(* CODESYS project FengHuang_PackBagbefore_V002.07.18.project

Project tree, tasks and I/O mapping:
  Device : AM403-CPU1608TN, Shenzhen Inovance Control Technology, version 3.5.11.10
      settings: PersistentStartAdddr = 0; PersistentStartEndAddr = 491519; Mode = 1
    application Application
      libraries: Standard, * (System); CmpHCAxisControl, 1.0.2.0 (Inovance); MEGA_Base, 0.0.0.1 (MEGA)
      task MainTask (cyclic, interval 16 ms, priority 1) calls Main
      task EIPSlaveServiceTask (cyclic, interval t#100ms, priority 30) calls EtherNetIPSlave.ServiceCycle
      task ETHERCAT (cyclic, interval 8 ms, priority 0) calls ETHERCAT.EtherCAT_Task, Call_Axis
      task EIPSlaveIOTask (cyclic, interval t#50ms, priority 1) calls EtherNetIPSlave.IOCycle
      DUTS/
        CT/
          data type ST_CT
        IO/
          data type EC6_0032A
          data type EC6_1616_Output
          data type EC6_3200A
          data type EC6_1616_Input
        HMI/
          data type ST_HMI_Vac_Pers
          data type ST_HMI_Cyl_Pers
          data type ST_HMI_Mac_Pers
          data type ST_HMI_Other
          data type ST_HMI_PrgVer
        Machine/
          data type ST_CardtSta
          data type ST_Machine
          data type ST_BagSta
        Data/
          data type ST_Data
        AXIS/
          data type ST_Ethercat
          data type Axis_POS
      FB/
        17_HMIFB/
          function block FB_Proface [ST]: ACT_Control, ACT_Empty, ACT_DummyCheck, ACT_Init
        16_VacuumFB/
          function block FB_Vacuum [ST]: ACT_Manual, ACT_Delay, ACT_Alarm, ACT_Output
        12_BlinkFB/
          data type ST_SysPulse
          function block FB_Blinker [ST]
        14_MachineFB/
          function block FB_Machine_1 [ST]: ACT_status, ACT_CT
          data type ST_OpeButton
          data type ST_DataMachine
          function block FB_Machine [ST]: ACT_Data, ACT_Start, ACT_Pause, ACT_Empty, ACT_Lamp, ACT_CycleTime, ACT_Stop, ACT_Init, ACT_General, ACT_Reset
        10_CylinderFB/
          function block FB_Cylinder [ST]: ACT_Delay, ACT_Output, ACT_Tip, ACT_Manual, ACT_Alarm
        05_StationFB/
          function block FB_Station [ST]: ACT_Init, ACT_State, ACT_Run, ACT_CycleTime, ACT_General
          data type E_State
        50_CycleTime/
          function block FB_CycleTime_2 [ST]
          function block FB_CycleTime_1 [ST]
          function block FB_CycleTime [ST]
        11_AxisFB/
          DUTs/
            data type ST_DataAxis
            data type ST_Axis_REF
          function block FB_Axis [ST]: ACT_Tip, ACT_Move, ACT_Reset, ACT_Halt, ACT_ReinitDrive, ACT_Home, ACT_Stop, ACT_Jog, ACT_Timeout, ACT_Power, ACT_Relative, ACT_InPos, ACT_Velocity, ACT_ReadStatus
      POUS/
        02_STATION/
          program S02_bowlFeeder [ST]: TipAuto, ILC, FlowAuto, TipManual, FlowInit, Alarm, Delay, General
          program S06_OpenBag [ST]: Delay, ILC, Alarm, FlowInit, TipManual, TipAuto, FlowAuto, General
          program S03_takebag [ST]: Delay, TipManual, FlowAuto, ILC, Alarm, General, FlowInit, TipAuto
          program S04_PushCard [ST]: Alarm, FlowInit, TipManual, General, ILC, FlowAuto, TipAuto, Delay
          program Add_distributor [ST]: ILC, Alarm, Delay, TipManual, TipAuto, General, FlowAuto, FlowInit
          program S01_transplant [ST]: TipManual, General, Delay, Alarm, TipAuto, FlowInit, ILC, FlowAuto
          program S05_CircleLine [ST]: Alarm, ILC, TipAuto, TipManual, General, Delay, FlowInit, FlowAuto
        01_LINK/
          program OUTPUT [ST]
          program INPUT [ST]
          program WLTLink [ST]
        03_CALL_standard/
          program ControlMachine [ST]: ACT_ALarm, ACT_Tip, ACT_Try_run, ACT_Count, ACT_InitDone, ACT_EIP_UP
          program Call_Axis [ST]: ACT_Link, ACT_Check
          program CallStandard [ST]: ACT_Machine, ACT_CT, ACT_Proface, ACT_Station, ACT_Blink, ACT_Cylinder, ACT_Vacuum
        program Main [ST]
      GVLS/
        global variables GVL_Standard
        global variables GVL_IO
        global variables GVL_Inside
      Symbols
      FC_check/
        function CheckDivLReal [ST]
        function CheckDivDInt [ST]
        function CheckLRangeUnsigned [ST]
        function CheckDivLInt [ST]
        function CheckRangeUnsigned [ST]
        function CheckRangeSigned [ST]
        function CheckLRangeSigned [ST]
        function CheckBounds [ST]
        function CheckDivReal [ST]
        function CheckPointer [ST]
      global variables PersistentVars
      trace CT (task ETHERCAT, trigger Positive on S05_CircleLine.Axis_Cycleline.rActVelo): S05_CircleLine.Axis_Cycleline.rActVelo
    HardWare Configuration
    ConfigStorage
    Network Configuration
      LocalBus Config
      EtherCAT Config
    Device Diagnosis
    GL10_3200END_1 : AM600-3200END, Inovance, version 00.00.00.10
        settings: ModuleBaseInfoStruct.BusType = 10; ModuleBaseInfoStruct.RackNumber = 1; ModuleBaseInfoStruct.SlotNumber = 2
        unmapped channels: IB(I), IB(II), IB(III), IB(IV)
    HwConfiguratioinDevice : SystemConfig, Inovance, version 00.00.00.10
        settings: NetworkConfigArray.NetworkConfigArray.BusType = 10; NetworkConfigArray.NetworkConfigArray.RackSum = 1; NetworkConfigArray.NetworkConfigArray.HardwareConfigArray.HardwareConfigArray.RackNo = 1; NetworkConfigArray.NetworkConfigArray.HardwareConfigArray.HardwareConfigArray.ModuleNum = 7; NetworkConfigArray.NetworkConfigArray.HardwareConfigArray.HardwareConfigArray.ModuleType.ModuleType = 40899; NetworkConfigArray.NetworkConfigArray.HardwareConfigArray.HardwareConfigArray.ModuleType.ModuleType = 40899; NetworkConfigArray.NetworkConfigArray.HardwareConfigArray.HardwareConfigArray.ModuleType.ModuleType = 40899; NetworkConfigArray.NetworkConfigArray.HardwareConfigArray.HardwareConfigArray.ModuleType.ModuleType = 40899; NetworkConfigArray.NetworkConfigArray.HardwareConfigArray.HardwareConfigArray.ModuleType.ModuleType = 45016; NetworkConfigArray.NetworkConfigArray.HardwareConfigArray.HardwareConfigArray.ModuleType.ModuleType = 45016; NetworkConfigArray.NetworkConfigArray.HardwareConfigArray.HardwareConfigArray.ModuleType.ModuleType = 45016; EnableFun = 1
    MODBUS_TCP : ModbusTCP Device, Inovance, version 00.00.00.10
    HIGH_SPEED_IO : High Speed IO Module, Inovance, version 00.00.00.20
        unmapped channels: InputData, OutputData
      HSIO
    GL10_3200END : AM600-3200END, Inovance, version 00.00.00.10
        settings: ModuleBaseInfoStruct.BusType = 10; ModuleBaseInfoStruct.RackNumber = 1; ModuleBaseInfoStruct.SlotNumber = 1
        unmapped channels: %IB2 IB(I), IB(II), IB(III), IB(IV)
    SoftMotion General Axis Pool
    GL10_0032ETN_1 : AM600-0032ETN, Inovance, version 00.00.00.10
        settings: ModuleBaseInfoStruct.BusType = 10; ModuleBaseInfoStruct.RackNumber = 1; ModuleBaseInfoStruct.SlotNumber = 6
        unmapped channels: QB(I), QB(II), QB(III), QB(IV)
    GL10_0032ETN_2 : AM600-0032ETN, Inovance, version 00.00.00.10
        settings: ModuleBaseInfoStruct.BusType = 10; ModuleBaseInfoStruct.RackNumber = 1; ModuleBaseInfoStruct.SlotNumber = 7
        unmapped channels: QB(I), QB(II), QB(III), QB(IV)
    GL10_3200END_2 : AM600-3200END, Inovance, version 00.00.00.10
        settings: ModuleBaseInfoStruct.BusType = 10; ModuleBaseInfoStruct.RackNumber = 1; ModuleBaseInfoStruct.SlotNumber = 3
        unmapped channels: IB(I), IB(II), IB(III), IB(IV)
    GL10_3200END_3 : AM600-3200END, Inovance, version 00.00.00.10
        settings: ModuleBaseInfoStruct.BusType = 10; ModuleBaseInfoStruct.RackNumber = 1; ModuleBaseInfoStruct.SlotNumber = 4
        unmapped channels: IB(I), IB(II), IB(III), IB(IV)
    GL10_0032ETN : AM600-0032ETN, Inovance, version 00.00.00.10
        settings: ModuleBaseInfoStruct.BusType = 10; ModuleBaseInfoStruct.RackNumber = 1; ModuleBaseInfoStruct.SlotNumber = 5
        unmapped channels: QB(I), QB(II), QB(III), QB(IV)
    ETHERCAT : EtherCAT Master SoftMotion, 3S - Smart Software Solutions GmbH, version 3.5.11.10
        settings:  = 0; MasterCycleTime = 8000; NetworkName = 'eth1'; SelectNetworkByName = TRUE; DisableTaskGeneration = True
      S03_supplybag_Y : SV660_1Axis_00911, Inovance, order no. InoSV660N, version Revision=16#00010000
          settings: FunCodeList = H02;H02-01;H02-02;H03;H03-03;H03-05;; WriteValueList = H02-01_8194_2_1_UINT_RW;H02-02_8194_3_1_UINT_RW;H03-03_8195_4_1_UINT_RW;H03-05_8195_6_1_UINT_RW;; Number of Outputs = 6; Number of Inputs = 10; Number of Infos about Outputs = 6; Number of Infos about Inputs = 10; StationAlias = 1001; Optional = False; DeviceIdenticationADO = 0; DeviceIdenticationMode = 0; Sync.Length = 18; Sync.Length = 32; FMMU.Length = 18; FMMU.Length = 32; AutoUpdate = False; DC sync0 cycletime = 8000; DC sync0 shift time = 0; DC sync1 cycletime = 8000; Number of SDO = 9; Homing method.Index = 16#6098; Homing method.Subindex = 16#00; Homing method.Value = 28; Homing method.Size = 8; Homing method.AbortIfError = FALSE; Homing method.JumpToLine = FALSE; Homing method.Line = 0; Homing method.CompleteAccess = FALSE; Speed during search for switch.Index = 16#6099; Speed during search for switch.Subindex = 16#01; Speed during search for switch.Value = 8388608; Speed during search for switch.Size = 32; Speed during search for switch.AbortIfError = FALSE; Speed during search for switch.JumpToLine = FALSE; Speed during search for switch.Line = 0; Speed during search for switch.CompleteAccess = FALSE; Homing acceleration.Index = 16#609A; Homing acceleration.Subindex = 16#00; Homing acceleration.Value = 419430400; Homing acceleration.Size = 32; Homing acceleration.AbortIfError = FALSE;
            Homing acceleration.JumpToLine = FALSE; Homing acceleration.Line = 0; Homing acceleration.CompleteAccess = FALSE; Speed during search for zero.Index = 16#6099; Speed during search for zero.Subindex = 16#02; Speed during search for zero.Value = 1677722; Speed during search for zero.Size = 32; Speed during search for zero.AbortIfError = FALSE; Speed during search for zero.JumpToLine = FALSE; Speed during search for zero.Line = 0; Speed during search for zero.CompleteAccess = FALSE; Time of home searching.Index = 16#2005; Time of home searching.Subindex = 16#24; Time of home searching.Value = 1500; Time of home searching.Size = 16; Time of home searching.AbortIfError = FALSE; Time of home searching.JumpToLine = FALSE; Time of home searching.Line = 0; Time of home searching.CompleteAccess = FALSE; Positive torque limit value.Index = 16#60E0; Positive torque limit value.Subindex = 16#00; Positive torque limit value.Value = 800; Positive torque limit value.Size = 16; Positive torque limit value.AbortIfError = FALSE; Positive torque limit value.JumpToLine = FALSE; Positive torque limit value.Line = 0; Positive torque limit value.CompleteAccess = FALSE; Negative torque limit value.Index = 16#60E1; Negative torque limit value.Subindex = 16#00; Negative torque limit value.Value = 800; Negative torque limit value.Size = 16; Negative torque limit value.AbortIfError = FALSE; Negative torque limit value.JumpToLine = FALSE; Negative torque limit value.Line = 0; Negative torque limit value.CompleteAccess = FALSE; Max profile velocity.Index = 16#607F; Max profile velocity.Subindex = 16#00; Max profile velocity.Value = 209715200; Max profile velocity.Size = 32; Max profile velocity.AbortIfError = FALSE;
            Max profile velocity.JumpToLine = FALSE; Max profile velocity.Line = 0; Max profile velocity.CompleteAccess = FALSE; RxTxPdo.NumberofEntries = 6; RxTxPdo.Sm = 2; Controlword.Index = 16#6040; Controlword.SubIndex = 0; Controlword.Size = 16; Controlword.DependOnSlot = false; Controlword.DependOnSlotGroup = false; Target position.Index = 16#607A; Target position.SubIndex = 0; Target position.Size = 32; Target position.DependOnSlot = false; Target position.DependOnSlotGroup = false; Touch probe function.Index = 16#60B8; Touch probe function.SubIndex = 0; Touch probe function.Size = 16; Touch probe function.DependOnSlot = false; Touch probe function.DependOnSlotGroup = false; Physical outputs.Index = 16#60FE; Physical outputs.SubIndex = 1; Physical outputs.Size = 32; Physical outputs.DependOnSlot = false; Physical outputs.DependOnSlotGroup = false; Target velocity.Index = 16#60FF; Target velocity.SubIndex = 0; Target velocity.Size = 32; Target velocity.DependOnSlot = false; Target velocity.DependOnSlotGroup = false; Target torque.Index = 16#6071; Target torque.SubIndex = 0; Target torque.Size = 16; Target torque.DependOnSlot = false; Target torque.DependOnSlotGroup = false; RxTxPdo.Sm = -1; RxTxPdo.NumberofEntries = 10; RxTxPdo.Sm = 3; Error code.Index = 16#603F; Error code.SubIndex = 0;
            Error code.Size = 16; Error code.DependOnSlot = false; Error code.DependOnSlotGroup = false; Statusword.Index = 16#6041; Statusword.SubIndex = 0; Statusword.Size = 16; Statusword.DependOnSlot = false; Statusword.DependOnSlotGroup = false; Position actual value.Index = 16#6064; Position actual value.SubIndex = 0; Position actual value.Size = 32; Position actual value.DependOnSlot = false; Position actual value.DependOnSlotGroup = false; Torque actual value.Index = 16#6077; Torque actual value.SubIndex = 0; Torque actual value.Size = 16; Torque actual value.DependOnSlot = false; Torque actual value.DependOnSlotGroup = false; Following error actual value.Index = 16#60F4; Following error actual value.SubIndex = 0; Following error actual value.Size = 32; Following error actual value.DependOnSlot = false; Following error actual value.DependOnSlotGroup = false; Touch probe status.Index = 16#60B9; Touch probe status.SubIndex = 0; Touch probe status.Size = 16; Touch probe status.DependOnSlot = false; Touch probe status.DependOnSlotGroup = false; Touch probe pos1 pos value.Index = 16#60BA; Touch probe pos1 pos value.SubIndex = 0; Touch probe pos1 pos value.Size = 32; Touch probe pos1 pos value.DependOnSlot = false; Touch probe pos1 pos value.DependOnSlotGroup = false; Touch probe pos2 pos value.Index = 16#60BC; Touch probe pos2 pos value.SubIndex = 0; Touch probe pos2 pos value.Size = 32; Touch probe pos2 pos value.DependOnSlot = false; Touch probe pos2 pos value.DependOnSlotGroup = false; Digital inputs.Index = 16#60FD; Digital inputs.SubIndex = 0;
            Digital inputs.Size = 32; Digital inputs.DependOnSlot = false; Digital inputs.DependOnSlotGroup = false; Velocity actual value.Index = 16#606C; Velocity actual value.SubIndex = 0; Velocity actual value.Size = 32; Velocity actual value.DependOnSlot = false; Velocity actual value.DependOnSlotGroup = false; RxTxPdo.Sm = -1; Controlword.Name = 'Controlword'; Controlword.DataType = 'UINT'; Target position.Name = 'Target position'; Target position.DataType = 'DINT'; Touch probe function.Name = 'Touch probe function'; Touch probe function.DataType = 'UINT'; Physical outputs.Name = 'Physical outputs'; Physical outputs.DataType = 'UDINT'; Target velocity.Name = 'Target velocity'; Target velocity.DataType = 'DINT'; Target torque.Name = 'Target torque'; Target torque.DataType = 'INT'; Error code.Name = 'Error code'; Error code.DataType = 'UINT'; Statusword.Name = 'Statusword'; Statusword.DataType = 'UINT'; Position actual value.Name = 'Position actual value'; Position actual value.DataType = 'DINT'; Torque actual value.Name = 'Torque actual value'; Torque actual value.DataType = 'INT'; Following error actual value.Name = 'Following error actual value'; Following error actual value.DataType = 'DINT'; Touch probe status.Name = 'Touch probe status'; Touch probe status.DataType = 'UINT'; Touch probe pos1 pos value.Name = 'Touch probe pos1 pos value'; Touch probe pos1 pos value.DataType = 'DINT'; Touch probe pos2 pos value.Name = 'Touch probe pos2 pos value'; Touch probe pos2 pos value.DataType = 'DINT'; Digital inputs.Name = 'Digital inputs'; Digital inputs.DataType = 'UDINT'; Velocity actual value.Name = 'Velocity actual value';
            Velocity actual value.DataType = 'DINT'
          unmapped channels: %QW500 Controlword, %QD251 Target position, %QW504 Touch probe function, %QD253 Physical outputs, Target velocity, Target torque, %IW500 Error code, %IW501 Statusword, %ID251 Position actual value, Torque actual value, Following error actual value, Touch probe status, Touch probe pos1 pos value, Touch probe pos2 pos value, Digital inputs, Velocity actual value
        Axis_4 : Axis, 3S - Smart Software Solutions GmbH, order no. 0, version 4.0.0.0
            settings: wDriveID = 3; dwRatioTechUnitsDenom = 2097152; iRatioTechUnitsNum = 5; 4000 = 1; 4001 = 0; 4003 = true; 4004 = 25; 4005 = 0; 4006 = 20; 4007 = 1000; 4008 = 4; 4009 = 1500; 4010 = 800; 4011 = 800; 4012 = 500; ScalingIncs = 16#800000; 6005 = 20; AdrOffset_8010 = 1000; BitOffset_8010 = 0; BitLength_8010 = 16; Address_8010 = '%QW500'; Type_8010 = 'UINT'; AddressPointer_8010 = ADR(%QW500); AdrOffset_8020 = 1004; BitOffset_8020 = 0; BitLength_8020 = 32; Address_8020 = '%QD251'; Type_8020 = 'DINT'; AddressPointer_8020 = ADR(%QD251); AdrOffset_8030 = 1016; BitOffset_8030 = 0; BitLength_8030 = 32; Address_8030 = '%QD254'; Type_8030 = 'DINT'; AddressPointer_8030 = ADR(%QD254); AdrOffset_8040 = 1020; BitOffset_8040 = 0; BitLength_8040 = 16; Address_8040 = '%QW510'; Type_8040 = 'INT';
              AddressPointer_8040 = ADR(%QW510); AdrOffset_8050 = 4294967295; BitOffset_8050 = 0; BitLength_8050 = 0; Address_8050 = ''; Type_8050 = ''; AddressPointer_8050 = 0; AdrOffset_8060 = 1008; BitOffset_8060 = 0; BitLength_8060 = 16; Address_8060 = '%QW504'; Type_8060 = 'UINT'; AddressPointer_8060 = ADR(%QW504); AdrOffset_8070 = 4294967295; BitOffset_8070 = 0; BitLength_8070 = 0; Address_8070 = ''; Type_8070 = ''; AddressPointer_8070 = 0; AdrOffset_8080 = 4294967295; BitOffset_8080 = 0; BitLength_8080 = 0; Address_8080 = ''; Type_8080 = ''; AddressPointer_8080 = 0; AdrOffset_8090 = 1012; BitOffset_8090 = 0; BitLength_8090 = 32; Address_8090 = '%QD253'; Type_8090 = 'UDINT'; AddressPointer_8090 = ADR(%QD253); AdrOffset_8510 = 1002; BitOffset_8510 = 0; BitLength_8510 = 16; Address_8510 = '%IW501'; Type_8510 = 'UINT'; AddressPointer_8510 = ADR(%IW501); AdrOffset_8520 = 1004; BitOffset_8520 = 0; BitLength_8520 = 32;
              Address_8520 = '%ID251'; Type_8520 = 'DINT'; AddressPointer_8520 = ADR(%ID251); AdrOffset_8530 = 1032; BitOffset_8530 = 0; BitLength_8530 = 32; Address_8530 = '%ID258'; Type_8530 = 'DINT'; AddressPointer_8530 = ADR(%ID258); AdrOffset_8540 = 1008; BitOffset_8540 = 0; BitLength_8540 = 16; Address_8540 = '%IW504'; Type_8540 = 'INT'; AddressPointer_8540 = ADR(%IW504); AdrOffset_8550 = 4294967295; BitOffset_8550 = 0; BitLength_8550 = 0; Address_8550 = ''; Type_8550 = ''; AddressPointer_8550 = 0; AdrOffset_8560 = 1028; BitOffset_8560 = 0; BitLength_8560 = 32; Address_8560 = '%ID257'; Type_8560 = 'UDINT'; AddressPointer_8560 = ADR(%ID257); AdrOffset_8570 = 1016; BitOffset_8570 = 0; BitLength_8570 = 16; Address_8570 = '%IW508'; Type_8570 = 'UINT'; AddressPointer_8570 = ADR(%IW508); AdrOffset_8580 = 1020; BitOffset_8580 = 0; BitLength_8580 = 32; Address_8580 = '%ID255'; Type_8580 = 'DINT'; AddressPointer_8580 = ADR(%ID255); AdrOffset_8590 = 4294967295;
              BitOffset_8590 = 0; BitLength_8590 = 0; Address_8590 = ''; Type_8590 = ''; AddressPointer_8590 = 0; AdrOffset_8600 = 1024; BitOffset_8600 = 0; BitLength_8600 = 32; Address_8600 = '%ID256'; Type_8600 = 'DINT'; AddressPointer_8600 = ADR(%ID256); AdrOffset_8600 = 4294967295; BitOffset_8600 = 0; BitLength_8600 = 0; Address_8610 = ''; Type_8610 = ''; AddressPointer_8610 = 0; AdrOffset_8620 = 1012; BitOffset_8620 = 0; BitLength_8620 = 32; Address_8620 = '%ID253'; Type_8620 = 'DINT'; AddressPointer_8620 = ADR(%ID253)
      Add_distributor_Y : SV660_1Axis_00911, Inovance, order no. InoSV660N, version Revision=16#00010000
          settings: FunCodeList = H02;H02-01;H03;H03-03;H03-05;; WriteValueList = H02-01_8194_2_1_UINT_RW;H03-03_8195_4_1_UINT_RW;H03-05_8195_6_1_UINT_RW;; Number of Outputs = 6; Number of Inputs = 10; Number of Infos about Outputs = 6; Number of Infos about Inputs = 10; Sync.Length = 18; Sync.Length = 32; FMMU.Length = 18; FMMU.Length = 32; AutoUpdate = False; DC sync0 cycletime = 8000; DC sync1 cycletime = 8000; Number of SDO = 9; Homing method.Index = 16#6098; Homing method.Subindex = 16#00; Homing method.Value = 28; Homing method.Size = 8; Homing method.AbortIfError = FALSE; Homing method.JumpToLine = FALSE; Homing method.Line = 0; Homing method.CompleteAccess = FALSE; Speed during search for switch.Index = 16#6099; Speed during search for switch.Subindex = 16#01; Speed during search for switch.Value = 8388608; Speed during search for switch.Size = 32; Speed during search for switch.AbortIfError = FALSE; Speed during search for switch.JumpToLine = FALSE; Speed during search for switch.Line = 0; Speed during search for switch.CompleteAccess = FALSE; Homing acceleration.Index = 16#609A; Homing acceleration.Subindex = 16#00; Homing acceleration.Value = 419430400; Homing acceleration.Size = 32; Homing acceleration.AbortIfError = FALSE; Homing acceleration.JumpToLine = FALSE; Homing acceleration.Line = 0; Homing acceleration.CompleteAccess = FALSE; Speed during search for zero.Index = 16#6099; Speed during search for zero.Subindex = 16#02;
            Speed during search for zero.Value = 1677722; Speed during search for zero.Size = 32; Speed during search for zero.AbortIfError = FALSE; Speed during search for zero.JumpToLine = FALSE; Speed during search for zero.Line = 0; Speed during search for zero.CompleteAccess = FALSE; Time of home searching.Index = 16#2005; Time of home searching.Subindex = 16#24; Time of home searching.Value = 1500; Time of home searching.Size = 16; Time of home searching.AbortIfError = FALSE; Time of home searching.JumpToLine = FALSE; Time of home searching.Line = 0; Time of home searching.CompleteAccess = FALSE; Positive torque limit value.Index = 16#60E0; Positive torque limit value.Subindex = 16#00; Positive torque limit value.Value = 800; Positive torque limit value.Size = 16; Positive torque limit value.AbortIfError = FALSE; Positive torque limit value.JumpToLine = FALSE; Positive torque limit value.Line = 0; Positive torque limit value.CompleteAccess = FALSE; Negative torque limit value.Index = 16#60E1; Negative torque limit value.Subindex = 16#00; Negative torque limit value.Value = 800; Negative torque limit value.Size = 16; Negative torque limit value.AbortIfError = FALSE; Negative torque limit value.JumpToLine = FALSE; Negative torque limit value.Line = 0; Negative torque limit value.CompleteAccess = FALSE; Max profile velocity.Index = 16#607F; Max profile velocity.Subindex = 16#00; Max profile velocity.Value = 209715200; Max profile velocity.Size = 32; Max profile velocity.AbortIfError = FALSE; Max profile velocity.JumpToLine = FALSE; Max profile velocity.Line = 0; Max profile velocity.CompleteAccess = FALSE; RxTxPdo.NumberofEntries = 6; RxTxPdo.Sm = 2;
            Controlword.Index = 16#6040; Controlword.SubIndex = 0; Controlword.Size = 16; Controlword.DependOnSlot = false; Controlword.DependOnSlotGroup = false; Target position.Index = 16#607A; Target position.SubIndex = 0; Target position.Size = 32; Target position.DependOnSlot = false; Target position.DependOnSlotGroup = false; Touch probe function.Index = 16#60B8; Touch probe function.SubIndex = 0; Touch probe function.Size = 16; Touch probe function.DependOnSlot = false; Touch probe function.DependOnSlotGroup = false; Physical outputs.Index = 16#60FE; Physical outputs.SubIndex = 1; Physical outputs.Size = 32; Physical outputs.DependOnSlot = false; Physical outputs.DependOnSlotGroup = false; Target velocity.Index = 16#60FF; Target velocity.SubIndex = 0; Target velocity.Size = 32; Target velocity.DependOnSlot = false; Target velocity.DependOnSlotGroup = false; Target torque.Index = 16#6071; Target torque.SubIndex = 0; Target torque.Size = 16; Target torque.DependOnSlot = false; Target torque.DependOnSlotGroup = false; RxTxPdo.Sm = -1; RxTxPdo.NumberofEntries = 10; RxTxPdo.Sm = 3; Error code.Index = 16#603F; Error code.SubIndex = 0; Error code.Size = 16; Error code.DependOnSlot = false; Error code.DependOnSlotGroup = false; Statusword.Index = 16#6041; Statusword.SubIndex = 0;
            Statusword.Size = 16; Statusword.DependOnSlot = false; Statusword.DependOnSlotGroup = false; Position actual value.Index = 16#6064; Position actual value.SubIndex = 0; Position actual value.Size = 32; Position actual value.DependOnSlot = false; Position actual value.DependOnSlotGroup = false; Torque actual value.Index = 16#6077; Torque actual value.SubIndex = 0; Torque actual value.Size = 16; Torque actual value.DependOnSlot = false; Torque actual value.DependOnSlotGroup = false; Following error actual value.Index = 16#60F4; Following error actual value.SubIndex = 0; Following error actual value.Size = 32; Following error actual value.DependOnSlot = false; Following error actual value.DependOnSlotGroup = false; Touch probe status.Index = 16#60B9; Touch probe status.SubIndex = 0; Touch probe status.Size = 16; Touch probe status.DependOnSlot = false; Touch probe status.DependOnSlotGroup = false; Touch probe pos1 pos value.Index = 16#60BA; Touch probe pos1 pos value.SubIndex = 0; Touch probe pos1 pos value.Size = 32; Touch probe pos1 pos value.DependOnSlot = false; Touch probe pos1 pos value.DependOnSlotGroup = false; Touch probe pos2 pos value.Index = 16#60BC; Touch probe pos2 pos value.SubIndex = 0; Touch probe pos2 pos value.Size = 32; Touch probe pos2 pos value.DependOnSlot = false; Touch probe pos2 pos value.DependOnSlotGroup = false; Digital inputs.Index = 16#60FD; Digital inputs.SubIndex = 0; Digital inputs.Size = 32; Digital inputs.DependOnSlot = false; Digital inputs.DependOnSlotGroup = false; Velocity actual value.Index = 16#606C; Velocity actual value.SubIndex = 0;
            Velocity actual value.Size = 32; Velocity actual value.DependOnSlot = false; Velocity actual value.DependOnSlotGroup = false; RxTxPdo.Sm = -1; Controlword.Name = 'Controlword'; Controlword.DataType = 'UINT'; Target position.Name = 'Target position'; Target position.DataType = 'DINT'; Touch probe function.Name = 'Touch probe function'; Touch probe function.DataType = 'UINT'; Physical outputs.Name = 'Physical outputs'; Physical outputs.DataType = 'UDINT'; Target velocity.Name = 'Target velocity'; Target velocity.DataType = 'DINT'; Target torque.Name = 'Target torque'; Target torque.DataType = 'INT'; Error code.Name = 'Error code'; Error code.DataType = 'UINT'; Statusword.Name = 'Statusword'; Statusword.DataType = 'UINT'; Position actual value.Name = 'Position actual value'; Position actual value.DataType = 'DINT'; Torque actual value.Name = 'Torque actual value'; Torque actual value.DataType = 'INT'; Following error actual value.Name = 'Following error actual value'; Following error actual value.DataType = 'DINT'; Touch probe status.Name = 'Touch probe status'; Touch probe status.DataType = 'UINT'; Touch probe pos1 pos value.Name = 'Touch probe pos1 pos value'; Touch probe pos1 pos value.DataType = 'DINT'; Touch probe pos2 pos value.Name = 'Touch probe pos2 pos value'; Touch probe pos2 pos value.DataType = 'DINT'; Digital inputs.Name = 'Digital inputs'; Digital inputs.DataType = 'UDINT'; Velocity actual value.Name = 'Velocity actual value'; Velocity actual value.DataType = 'DINT'
          unmapped channels: %QW560 Controlword, Target position, Touch probe function, Physical outputs, Target velocity, Target torque, %IW560 Error code, Statusword, Position actual value, Torque actual value, Following error actual value, Touch probe status, Touch probe pos1 pos value, Touch probe pos2 pos value, Digital inputs, Velocity actual value
        Axis_1 : Axis, 3S - Smart Software Solutions GmbH, order no. 0, version 4.0.0.0
            settings: wDriveID = 0; dwRatioTechUnitsDenom = 2097152; iRatioTechUnitsNum = 5; 4000 = 1; 4001 = 0; 4003 = true; 4004 = 25; 4005 = 0; 4006 = 20; 4007 = 1000; 4008 = 4; 4009 = 1500; 4010 = 800; 4011 = 800; 4012 = 500; ScalingIncs = 16#800000; 6005 = 20; AdrOffset_8010 = 1120; BitOffset_8010 = 0; BitLength_8010 = 16; Address_8010 = '%QW560'; Type_8010 = 'UINT'; AddressPointer_8010 = ADR(%QW560); AdrOffset_8020 = 1124; BitOffset_8020 = 0; BitLength_8020 = 32; Address_8020 = '%QD281'; Type_8020 = 'DINT'; AddressPointer_8020 = ADR(%QD281); AdrOffset_8030 = 1136; BitOffset_8030 = 0; BitLength_8030 = 32; Address_8030 = '%QD284'; Type_8030 = 'DINT'; AddressPointer_8030 = ADR(%QD284); AdrOffset_8040 = 1140; BitOffset_8040 = 0; BitLength_8040 = 16; Address_8040 = '%QW570'; Type_8040 = 'INT';
              AddressPointer_8040 = ADR(%QW570); AdrOffset_8050 = 4294967295; BitOffset_8050 = 0; BitLength_8050 = 0; Address_8050 = ''; Type_8050 = ''; AddressPointer_8050 = 0; AdrOffset_8060 = 1128; BitOffset_8060 = 0; BitLength_8060 = 16; Address_8060 = '%QW564'; Type_8060 = 'UINT'; AddressPointer_8060 = ADR(%QW564); AdrOffset_8070 = 4294967295; BitOffset_8070 = 0; BitLength_8070 = 0; Address_8070 = ''; Type_8070 = ''; AddressPointer_8070 = 0; AdrOffset_8080 = 4294967295; BitOffset_8080 = 0; BitLength_8080 = 0; Address_8080 = ''; Type_8080 = ''; AddressPointer_8080 = 0; AdrOffset_8090 = 1132; BitOffset_8090 = 0; BitLength_8090 = 32; Address_8090 = '%QD283'; Type_8090 = 'UDINT'; AddressPointer_8090 = ADR(%QD283); AdrOffset_8510 = 1122; BitOffset_8510 = 0; BitLength_8510 = 16; Address_8510 = '%IW561'; Type_8510 = 'UINT'; AddressPointer_8510 = ADR(%IW561); AdrOffset_8520 = 1124; BitOffset_8520 = 0; BitLength_8520 = 32;
              Address_8520 = '%ID281'; Type_8520 = 'DINT'; AddressPointer_8520 = ADR(%ID281); AdrOffset_8530 = 1152; BitOffset_8530 = 0; BitLength_8530 = 32; Address_8530 = '%ID288'; Type_8530 = 'DINT'; AddressPointer_8530 = ADR(%ID288); AdrOffset_8540 = 1128; BitOffset_8540 = 0; BitLength_8540 = 16; Address_8540 = '%IW564'; Type_8540 = 'INT'; AddressPointer_8540 = ADR(%IW564); AdrOffset_8550 = 4294967295; BitOffset_8550 = 0; BitLength_8550 = 0; Address_8550 = ''; Type_8550 = ''; AddressPointer_8550 = 0; AdrOffset_8560 = 1148; BitOffset_8560 = 0; BitLength_8560 = 32; Address_8560 = '%ID287'; Type_8560 = 'UDINT'; AddressPointer_8560 = ADR(%ID287); AdrOffset_8570 = 1136; BitOffset_8570 = 0; BitLength_8570 = 16; Address_8570 = '%IW568'; Type_8570 = 'UINT'; AddressPointer_8570 = ADR(%IW568); AdrOffset_8580 = 1140; BitOffset_8580 = 0; BitLength_8580 = 32; Address_8580 = '%ID285'; Type_8580 = 'DINT'; AddressPointer_8580 = ADR(%ID285); AdrOffset_8590 = 4294967295;
              BitOffset_8590 = 0; BitLength_8590 = 0; Address_8590 = ''; Type_8590 = ''; AddressPointer_8590 = 0; AdrOffset_8600 = 1144; BitOffset_8600 = 0; BitLength_8600 = 32; Address_8600 = '%ID286'; Type_8600 = 'DINT'; AddressPointer_8600 = ADR(%ID286); AdrOffset_8600 = 4294967295; BitOffset_8600 = 0; BitLength_8600 = 0; Address_8610 = ''; Type_8610 = ''; AddressPointer_8610 = 0; AdrOffset_8620 = 1132; BitOffset_8620 = 0; BitLength_8620 = 32; Address_8620 = '%ID283'; Type_8620 = 'DINT'; AddressPointer_8620 = ADR(%ID283)
      S03_CycleLine : SV660_1Axis_00911, Inovance, order no. InoSV660N, version Revision=16#00010000
          settings: FunCodeList = H02;H02-02;H0D;H0D-20;; WriteValueList = H02-02_8194_3_0_UINT_RW;H0D-20_8205_21_1_UINT_RW;; Number of Outputs = 6; Number of Inputs = 10; Number of Infos about Outputs = 6; Number of Infos about Inputs = 10; Sync.Length = 18; Sync.Length = 32; FMMU.Length = 18; FMMU.Length = 32; AutoUpdate = False; DC sync0 cycletime = 8000; DC sync1 cycletime = 8000; Number of SDO = 9; Homing method.Index = 16#6098; Homing method.Subindex = 16#00; Homing method.Value = 20; Homing method.Size = 8; Homing method.AbortIfError = FALSE; Homing method.JumpToLine = FALSE; Homing method.Line = 0; Homing method.CompleteAccess = FALSE; Speed during search for switch.Index = 16#6099; Speed during search for switch.Subindex = 16#01; Speed during search for switch.Value = 4194304; Speed during search for switch.Size = 32; Speed during search for switch.AbortIfError = FALSE; Speed during search for switch.JumpToLine = FALSE; Speed during search for switch.Line = 0; Speed during search for switch.CompleteAccess = FALSE; Homing acceleration.Index = 16#609A; Homing acceleration.Subindex = 16#00; Homing acceleration.Value = 209715200; Homing acceleration.Size = 32; Homing acceleration.AbortIfError = FALSE; Homing acceleration.JumpToLine = FALSE; Homing acceleration.Line = 0; Homing acceleration.CompleteAccess = FALSE; Speed during search for zero.Index = 16#6099; Speed during search for zero.Subindex = 16#02;
            Speed during search for zero.Value = 838861; Speed during search for zero.Size = 32; Speed during search for zero.AbortIfError = FALSE; Speed during search for zero.JumpToLine = FALSE; Speed during search for zero.Line = 0; Speed during search for zero.CompleteAccess = FALSE; Time of home searching.Index = 16#2005; Time of home searching.Subindex = 16#24; Time of home searching.Value = 1500; Time of home searching.Size = 16; Time of home searching.AbortIfError = FALSE; Time of home searching.JumpToLine = FALSE; Time of home searching.Line = 0; Time of home searching.CompleteAccess = FALSE; Positive torque limit value.Index = 16#60E0; Positive torque limit value.Subindex = 16#00; Positive torque limit value.Value = 800; Positive torque limit value.Size = 16; Positive torque limit value.AbortIfError = FALSE; Positive torque limit value.JumpToLine = FALSE; Positive torque limit value.Line = 0; Positive torque limit value.CompleteAccess = FALSE; Negative torque limit value.Index = 16#60E1; Negative torque limit value.Subindex = 16#00; Negative torque limit value.Value = 800; Negative torque limit value.Size = 16; Negative torque limit value.AbortIfError = FALSE; Negative torque limit value.JumpToLine = FALSE; Negative torque limit value.Line = 0; Negative torque limit value.CompleteAccess = FALSE; Max profile velocity.Index = 16#607F; Max profile velocity.Subindex = 16#00; Max profile velocity.Value = 104857600; Max profile velocity.Size = 32; Max profile velocity.AbortIfError = FALSE; Max profile velocity.JumpToLine = FALSE; Max profile velocity.Line = 0; Max profile velocity.CompleteAccess = FALSE; RxTxPdo.NumberofEntries = 6; RxTxPdo.Sm = 2;
            Controlword.Index = 16#6040; Controlword.SubIndex = 0; Controlword.Size = 16; Controlword.DependOnSlot = false; Controlword.DependOnSlotGroup = false; Target position.Index = 16#607A; Target position.SubIndex = 0; Target position.Size = 32; Target position.DependOnSlot = false; Target position.DependOnSlotGroup = false; Touch probe function.Index = 16#60B8; Touch probe function.SubIndex = 0; Touch probe function.Size = 16; Touch probe function.DependOnSlot = false; Touch probe function.DependOnSlotGroup = false; Physical outputs.Index = 16#60FE; Physical outputs.SubIndex = 1; Physical outputs.Size = 32; Physical outputs.DependOnSlot = false; Physical outputs.DependOnSlotGroup = false; Target velocity.Index = 16#60FF; Target velocity.SubIndex = 0; Target velocity.Size = 32; Target velocity.DependOnSlot = false; Target velocity.DependOnSlotGroup = false; Target torque.Index = 16#6071; Target torque.SubIndex = 0; Target torque.Size = 16; Target torque.DependOnSlot = false; Target torque.DependOnSlotGroup = false; RxTxPdo.Sm = -1; RxTxPdo.NumberofEntries = 10; RxTxPdo.Sm = 3; Error code.Index = 16#603F; Error code.SubIndex = 0; Error code.Size = 16; Error code.DependOnSlot = false; Error code.DependOnSlotGroup = false; Statusword.Index = 16#6041; Statusword.SubIndex = 0;
            Statusword.Size = 16; Statusword.DependOnSlot = false; Statusword.DependOnSlotGroup = false; Position actual value.Index = 16#6064; Position actual value.SubIndex = 0; Position actual value.Size = 32; Position actual value.DependOnSlot = false; Position actual value.DependOnSlotGroup = false; Torque actual value.Index = 16#6077; Torque actual value.SubIndex = 0; Torque actual value.Size = 16; Torque actual value.DependOnSlot = false; Torque actual value.DependOnSlotGroup = false; Following error actual value.Index = 16#60F4; Following error actual value.SubIndex = 0; Following error actual value.Size = 32; Following error actual value.DependOnSlot = false; Following error actual value.DependOnSlotGroup = false; Touch probe status.Index = 16#60B9; Touch probe status.SubIndex = 0; Touch probe status.Size = 16; Touch probe status.DependOnSlot = false; Touch probe status.DependOnSlotGroup = false; Touch probe pos1 pos value.Index = 16#60BA; Touch probe pos1 pos value.SubIndex = 0; Touch probe pos1 pos value.Size = 32; Touch probe pos1 pos value.DependOnSlot = false; Touch probe pos1 pos value.DependOnSlotGroup = false; Touch probe pos2 pos value.Index = 16#60BC; Touch probe pos2 pos value.SubIndex = 0; Touch probe pos2 pos value.Size = 32; Touch probe pos2 pos value.DependOnSlot = false; Touch probe pos2 pos value.DependOnSlotGroup = false; Digital inputs.Index = 16#60FD; Digital inputs.SubIndex = 0; Digital inputs.Size = 32; Digital inputs.DependOnSlot = false; Digital inputs.DependOnSlotGroup = false; Velocity actual value.Index = 16#606C; Velocity actual value.SubIndex = 0;
            Velocity actual value.Size = 32; Velocity actual value.DependOnSlot = false; Velocity actual value.DependOnSlotGroup = false; RxTxPdo.Sm = -1; Controlword.Name = 'Controlword'; Controlword.DataType = 'UINT'; Target position.Name = 'Target position'; Target position.DataType = 'DINT'; Touch probe function.Name = 'Touch probe function'; Touch probe function.DataType = 'UINT'; Physical outputs.Name = 'Physical outputs'; Physical outputs.DataType = 'UDINT'; Target velocity.Name = 'Target velocity'; Target velocity.DataType = 'DINT'; Target torque.Name = 'Target torque'; Target torque.DataType = 'INT'; Error code.Name = 'Error code'; Error code.DataType = 'UINT'; Statusword.Name = 'Statusword'; Statusword.DataType = 'UINT'; Position actual value.Name = 'Position actual value'; Position actual value.DataType = 'DINT'; Torque actual value.Name = 'Torque actual value'; Torque actual value.DataType = 'INT'; Following error actual value.Name = 'Following error actual value'; Following error actual value.DataType = 'DINT'; Touch probe status.Name = 'Touch probe status'; Touch probe status.DataType = 'UINT'; Touch probe pos1 pos value.Name = 'Touch probe pos1 pos value'; Touch probe pos1 pos value.DataType = 'DINT'; Touch probe pos2 pos value.Name = 'Touch probe pos2 pos value'; Touch probe pos2 pos value.DataType = 'DINT'; Digital inputs.Name = 'Digital inputs'; Digital inputs.DataType = 'UDINT'; Velocity actual value.Name = 'Velocity actual value'; Velocity actual value.DataType = 'DINT'
          unmapped channels: %QW600 Controlword, Target position, Touch probe function, Physical outputs, Target velocity, Target torque, %IW600 Error code, Statusword, Position actual value, Torque actual value, Following error actual value, Touch probe status, Touch probe pos1 pos value, Touch probe pos2 pos value, Digital inputs, Velocity actual value
        Axis_3 : Axis, 3S - Smart Software Solutions GmbH, order no. 0, version 4.0.0.0
            settings: wDriveID = 2; dwRatioTechUnitsDenom = 1048576; iRatioTechUnitsNum = 5; 4000 = 1; 4001 = 1; 4003 = true; 4004 = 17; 4005 = 0; 4006 = 20; 4007 = 1000; 4008 = 4; 4009 = 1500; 4010 = 800; 4011 = 800; 4012 = 500; ScalingIncs = 16#800000; ScalingMotorTurns2 = 5; 6005 = 200; AdrOffset_8010 = 1200; BitOffset_8010 = 0; BitLength_8010 = 16; Address_8010 = '%QW600'; Type_8010 = 'UINT'; AddressPointer_8010 = ADR(%QW600); AdrOffset_8020 = 1204; BitOffset_8020 = 0; BitLength_8020 = 32; Address_8020 = '%QD301'; Type_8020 = 'DINT'; AddressPointer_8020 = ADR(%QD301); AdrOffset_8030 = 1216; BitOffset_8030 = 0; BitLength_8030 = 32; Address_8030 = '%QD304'; Type_8030 = 'DINT'; AddressPointer_8030 = ADR(%QD304); AdrOffset_8040 = 1220; BitOffset_8040 = 0; BitLength_8040 = 16; Address_8040 = '%QW610';
              Type_8040 = 'INT'; AddressPointer_8040 = ADR(%QW610); AdrOffset_8050 = 4294967295; BitOffset_8050 = 0; BitLength_8050 = 0; Address_8050 = ''; Type_8050 = ''; AddressPointer_8050 = 0; AdrOffset_8060 = 1208; BitOffset_8060 = 0; BitLength_8060 = 16; Address_8060 = '%QW604'; Type_8060 = 'UINT'; AddressPointer_8060 = ADR(%QW604); AdrOffset_8070 = 4294967295; BitOffset_8070 = 0; BitLength_8070 = 0; Address_8070 = ''; Type_8070 = ''; AddressPointer_8070 = 0; AdrOffset_8080 = 4294967295; BitOffset_8080 = 0; BitLength_8080 = 0; Address_8080 = ''; Type_8080 = ''; AddressPointer_8080 = 0; AdrOffset_8090 = 1212; BitOffset_8090 = 0; BitLength_8090 = 32; Address_8090 = '%QD303'; Type_8090 = 'UDINT'; AddressPointer_8090 = ADR(%QD303); AdrOffset_8510 = 1202; BitOffset_8510 = 0; BitLength_8510 = 16; Address_8510 = '%IW601'; Type_8510 = 'UINT'; AddressPointer_8510 = ADR(%IW601); AdrOffset_8520 = 1204; BitOffset_8520 = 0;
              BitLength_8520 = 32; Address_8520 = '%ID301'; Type_8520 = 'DINT'; AddressPointer_8520 = ADR(%ID301); AdrOffset_8530 = 1232; BitOffset_8530 = 0; BitLength_8530 = 32; Address_8530 = '%ID308'; Type_8530 = 'DINT'; AddressPointer_8530 = ADR(%ID308); AdrOffset_8540 = 1208; BitOffset_8540 = 0; BitLength_8540 = 16; Address_8540 = '%IW604'; Type_8540 = 'INT'; AddressPointer_8540 = ADR(%IW604); AdrOffset_8550 = 4294967295; BitOffset_8550 = 0; BitLength_8550 = 0; Address_8550 = ''; Type_8550 = ''; AddressPointer_8550 = 0; AdrOffset_8560 = 1228; BitOffset_8560 = 0; BitLength_8560 = 32; Address_8560 = '%ID307'; Type_8560 = 'UDINT'; AddressPointer_8560 = ADR(%ID307); AdrOffset_8570 = 1216; BitOffset_8570 = 0; BitLength_8570 = 16; Address_8570 = '%IW608'; Type_8570 = 'UINT'; AddressPointer_8570 = ADR(%IW608); AdrOffset_8580 = 1220; BitOffset_8580 = 0; BitLength_8580 = 32; Address_8580 = '%ID305'; Type_8580 = 'DINT'; AddressPointer_8580 = ADR(%ID305);
              AdrOffset_8590 = 4294967295; BitOffset_8590 = 0; BitLength_8590 = 0; Address_8590 = ''; Type_8590 = ''; AddressPointer_8590 = 0; AdrOffset_8600 = 1224; BitOffset_8600 = 0; BitLength_8600 = 32; Address_8600 = '%ID306'; Type_8600 = 'DINT'; AddressPointer_8600 = ADR(%ID306); AdrOffset_8600 = 4294967295; BitOffset_8600 = 0; BitLength_8600 = 0; Address_8610 = ''; Type_8610 = ''; AddressPointer_8610 = 0; AdrOffset_8620 = 1212; BitOffset_8620 = 0; BitLength_8620 = 32; Address_8620 = '%ID303'; Type_8620 = 'DINT'; AddressPointer_8620 = ADR(%ID303)
      S01_CycleLine : SV660_1Axis_00911, Inovance, order no. InoSV660N, version Revision=16#00010000
          settings: FunCodeList = H02;H02-02;H03;H03-03;H03-05;H0D;H0D-20;; WriteValueList = H02-02_8194_3_1_UINT_RW;H03-03_8195_4_0_UINT_RW;H03-05_8195_6_0_UINT_RW;H0D-20_8205_21_0_UINT_RW;; Number of Outputs = 6; Number of Inputs = 10; Number of Infos about Outputs = 6; Number of Infos about Inputs = 10; Sync.Length = 18; Sync.Length = 32; FMMU.Length = 18; FMMU.Length = 32; AutoUpdate = False; DC sync0 cycletime = 8000; DC sync1 cycletime = 8000; Number of SDO = 9; Homing method.Index = 16#6098; Homing method.Subindex = 16#00; Homing method.Value = 20; Homing method.Size = 8; Homing method.AbortIfError = FALSE; Homing method.JumpToLine = FALSE; Homing method.Line = 0; Homing method.CompleteAccess = FALSE; Speed during search for switch.Index = 16#6099; Speed during search for switch.Subindex = 16#01; Speed during search for switch.Value = 4194304; Speed during search for switch.Size = 32; Speed during search for switch.AbortIfError = FALSE; Speed during search for switch.JumpToLine = FALSE; Speed during search for switch.Line = 0; Speed during search for switch.CompleteAccess = FALSE; Homing acceleration.Index = 16#609A; Homing acceleration.Subindex = 16#00; Homing acceleration.Value = 209715200; Homing acceleration.Size = 32; Homing acceleration.AbortIfError = FALSE; Homing acceleration.JumpToLine = FALSE; Homing acceleration.Line = 0; Homing acceleration.CompleteAccess = FALSE; Speed during search for zero.Index = 16#6099; Speed during search for zero.Subindex = 16#02;
            Speed during search for zero.Value = 838861; Speed during search for zero.Size = 32; Speed during search for zero.AbortIfError = FALSE; Speed during search for zero.JumpToLine = FALSE; Speed during search for zero.Line = 0; Speed during search for zero.CompleteAccess = FALSE; Time of home searching.Index = 16#2005; Time of home searching.Subindex = 16#24; Time of home searching.Value = 1500; Time of home searching.Size = 16; Time of home searching.AbortIfError = FALSE; Time of home searching.JumpToLine = FALSE; Time of home searching.Line = 0; Time of home searching.CompleteAccess = FALSE; Positive torque limit value.Index = 16#60E0; Positive torque limit value.Subindex = 16#00; Positive torque limit value.Value = 800; Positive torque limit value.Size = 16; Positive torque limit value.AbortIfError = FALSE; Positive torque limit value.JumpToLine = FALSE; Positive torque limit value.Line = 0; Positive torque limit value.CompleteAccess = FALSE; Negative torque limit value.Index = 16#60E1; Negative torque limit value.Subindex = 16#00; Negative torque limit value.Value = 800; Negative torque limit value.Size = 16; Negative torque limit value.AbortIfError = FALSE; Negative torque limit value.JumpToLine = FALSE; Negative torque limit value.Line = 0; Negative torque limit value.CompleteAccess = FALSE; Max profile velocity.Index = 16#607F; Max profile velocity.Subindex = 16#00; Max profile velocity.Value = 104857600; Max profile velocity.Size = 32; Max profile velocity.AbortIfError = FALSE; Max profile velocity.JumpToLine = FALSE; Max profile velocity.Line = 0; Max profile velocity.CompleteAccess = FALSE; RxTxPdo.NumberofEntries = 6; RxTxPdo.Sm = 2;
            Controlword.Index = 16#6040; Controlword.SubIndex = 0; Controlword.Size = 16; Controlword.DependOnSlot = false; Controlword.DependOnSlotGroup = false; Target position.Index = 16#607A; Target position.SubIndex = 0; Target position.Size = 32; Target position.DependOnSlot = false; Target position.DependOnSlotGroup = false; Touch probe function.Index = 16#60B8; Touch probe function.SubIndex = 0; Touch probe function.Size = 16; Touch probe function.DependOnSlot = false; Touch probe function.DependOnSlotGroup = false; Physical outputs.Index = 16#60FE; Physical outputs.SubIndex = 1; Physical outputs.Size = 32; Physical outputs.DependOnSlot = false; Physical outputs.DependOnSlotGroup = false; Target velocity.Index = 16#60FF; Target velocity.SubIndex = 0; Target velocity.Size = 32; Target velocity.DependOnSlot = false; Target velocity.DependOnSlotGroup = false; Target torque.Index = 16#6071; Target torque.SubIndex = 0; Target torque.Size = 16; Target torque.DependOnSlot = false; Target torque.DependOnSlotGroup = false; RxTxPdo.Sm = -1; RxTxPdo.NumberofEntries = 10; RxTxPdo.Sm = 3; Error code.Index = 16#603F; Error code.SubIndex = 0; Error code.Size = 16; Error code.DependOnSlot = false; Error code.DependOnSlotGroup = false; Statusword.Index = 16#6041; Statusword.SubIndex = 0;
            Statusword.Size = 16; Statusword.DependOnSlot = false; Statusword.DependOnSlotGroup = false; Position actual value.Index = 16#6064; Position actual value.SubIndex = 0; Position actual value.Size = 32; Position actual value.DependOnSlot = false; Position actual value.DependOnSlotGroup = false; Torque actual value.Index = 16#6077; Torque actual value.SubIndex = 0; Torque actual value.Size = 16; Torque actual value.DependOnSlot = false; Torque actual value.DependOnSlotGroup = false; Following error actual value.Index = 16#60F4; Following error actual value.SubIndex = 0; Following error actual value.Size = 32; Following error actual value.DependOnSlot = false; Following error actual value.DependOnSlotGroup = false; Touch probe status.Index = 16#60B9; Touch probe status.SubIndex = 0; Touch probe status.Size = 16; Touch probe status.DependOnSlot = false; Touch probe status.DependOnSlotGroup = false; Touch probe pos1 pos value.Index = 16#60BA; Touch probe pos1 pos value.SubIndex = 0; Touch probe pos1 pos value.Size = 32; Touch probe pos1 pos value.DependOnSlot = false; Touch probe pos1 pos value.DependOnSlotGroup = false; Touch probe pos2 pos value.Index = 16#60BC; Touch probe pos2 pos value.SubIndex = 0; Touch probe pos2 pos value.Size = 32; Touch probe pos2 pos value.DependOnSlot = false; Touch probe pos2 pos value.DependOnSlotGroup = false; Digital inputs.Index = 16#60FD; Digital inputs.SubIndex = 0; Digital inputs.Size = 32; Digital inputs.DependOnSlot = false; Digital inputs.DependOnSlotGroup = false; Velocity actual value.Index = 16#606C; Velocity actual value.SubIndex = 0;
            Velocity actual value.Size = 32; Velocity actual value.DependOnSlot = false; Velocity actual value.DependOnSlotGroup = false; RxTxPdo.Sm = -1; Controlword.Name = 'Controlword'; Controlword.DataType = 'UINT'; Target position.Name = 'Target position'; Target position.DataType = 'DINT'; Touch probe function.Name = 'Touch probe function'; Touch probe function.DataType = 'UINT'; Physical outputs.Name = 'Physical outputs'; Physical outputs.DataType = 'UDINT'; Target velocity.Name = 'Target velocity'; Target velocity.DataType = 'DINT'; Target torque.Name = 'Target torque'; Target torque.DataType = 'INT'; Error code.Name = 'Error code'; Error code.DataType = 'UINT'; Statusword.Name = 'Statusword'; Statusword.DataType = 'UINT'; Position actual value.Name = 'Position actual value'; Position actual value.DataType = 'DINT'; Torque actual value.Name = 'Torque actual value'; Torque actual value.DataType = 'INT'; Following error actual value.Name = 'Following error actual value'; Following error actual value.DataType = 'DINT'; Touch probe status.Name = 'Touch probe status'; Touch probe status.DataType = 'UINT'; Touch probe pos1 pos value.Name = 'Touch probe pos1 pos value'; Touch probe pos1 pos value.DataType = 'DINT'; Touch probe pos2 pos value.Name = 'Touch probe pos2 pos value'; Touch probe pos2 pos value.DataType = 'DINT'; Digital inputs.Name = 'Digital inputs'; Digital inputs.DataType = 'UDINT'; Velocity actual value.Name = 'Velocity actual value'; Velocity actual value.DataType = 'DINT'
          unmapped channels: %QW580 Controlword, Target position, Touch probe function, Physical outputs, Target velocity, Target torque, %IW580 Error code, Statusword, Position actual value, Torque actual value, Following error actual value, Touch probe status, Touch probe pos1 pos value, Touch probe pos2 pos value, Digital inputs, Velocity actual value
        Axis_2 : Axis, 3S - Smart Software Solutions GmbH, order no. 0, version 4.0.0.0
            settings: dwRatioTechUnitsDenom = 1048576; iRatioTechUnitsNum = 5; 4000 = 1; 4001 = 1; 4003 = true; 4004 = 17; 4005 = 0; 4006 = 20; 4007 = 1000; 4008 = 4; 4009 = 1500; 4010 = 800; 4011 = 800; 4012 = 500; ScalingIncs = 16#800000; ScalingMotorTurns2 = 5; 6005 = 200; AdrOffset_8010 = 1160; BitOffset_8010 = 0; BitLength_8010 = 16; Address_8010 = '%QW580'; Type_8010 = 'UINT'; AddressPointer_8010 = ADR(%QW580); AdrOffset_8020 = 1164; BitOffset_8020 = 0; BitLength_8020 = 32; Address_8020 = '%QD291'; Type_8020 = 'DINT'; AddressPointer_8020 = ADR(%QD291); AdrOffset_8030 = 1176; BitOffset_8030 = 0; BitLength_8030 = 32; Address_8030 = '%QD294'; Type_8030 = 'DINT'; AddressPointer_8030 = ADR(%QD294); AdrOffset_8040 = 1180; BitOffset_8040 = 0; BitLength_8040 = 16; Address_8040 = '%QW590'; Type_8040 = 'INT';
              AddressPointer_8040 = ADR(%QW590); AdrOffset_8050 = 4294967295; BitOffset_8050 = 0; BitLength_8050 = 0; Address_8050 = ''; Type_8050 = ''; AddressPointer_8050 = 0; AdrOffset_8060 = 1168; BitOffset_8060 = 0; BitLength_8060 = 16; Address_8060 = '%QW584'; Type_8060 = 'UINT'; AddressPointer_8060 = ADR(%QW584); AdrOffset_8070 = 4294967295; BitOffset_8070 = 0; BitLength_8070 = 0; Address_8070 = ''; Type_8070 = ''; AddressPointer_8070 = 0; AdrOffset_8080 = 4294967295; BitOffset_8080 = 0; BitLength_8080 = 0; Address_8080 = ''; Type_8080 = ''; AddressPointer_8080 = 0; AdrOffset_8090 = 1172; BitOffset_8090 = 0; BitLength_8090 = 32; Address_8090 = '%QD293'; Type_8090 = 'UDINT'; AddressPointer_8090 = ADR(%QD293); AdrOffset_8510 = 1162; BitOffset_8510 = 0; BitLength_8510 = 16; Address_8510 = '%IW581'; Type_8510 = 'UINT'; AddressPointer_8510 = ADR(%IW581); AdrOffset_8520 = 1164; BitOffset_8520 = 0; BitLength_8520 = 32;
              Address_8520 = '%ID291'; Type_8520 = 'DINT'; AddressPointer_8520 = ADR(%ID291); AdrOffset_8530 = 1192; BitOffset_8530 = 0; BitLength_8530 = 32; Address_8530 = '%ID298'; Type_8530 = 'DINT'; AddressPointer_8530 = ADR(%ID298); AdrOffset_8540 = 1168; BitOffset_8540 = 0; BitLength_8540 = 16; Address_8540 = '%IW584'; Type_8540 = 'INT'; AddressPointer_8540 = ADR(%IW584); AdrOffset_8550 = 4294967295; BitOffset_8550 = 0; BitLength_8550 = 0; Address_8550 = ''; Type_8550 = ''; AddressPointer_8550 = 0; AdrOffset_8560 = 1188; BitOffset_8560 = 0; BitLength_8560 = 32; Address_8560 = '%ID297'; Type_8560 = 'UDINT'; AddressPointer_8560 = ADR(%ID297); AdrOffset_8570 = 1176; BitOffset_8570 = 0; BitLength_8570 = 16; Address_8570 = '%IW588'; Type_8570 = 'UINT'; AddressPointer_8570 = ADR(%IW588); AdrOffset_8580 = 1180; BitOffset_8580 = 0; BitLength_8580 = 32; Address_8580 = '%ID295'; Type_8580 = 'DINT'; AddressPointer_8580 = ADR(%ID295); AdrOffset_8590 = 4294967295;
              BitOffset_8590 = 0; BitLength_8590 = 0; Address_8590 = ''; Type_8590 = ''; AddressPointer_8590 = 0; AdrOffset_8600 = 1184; BitOffset_8600 = 0; BitLength_8600 = 32; Address_8600 = '%ID296'; Type_8600 = 'DINT'; AddressPointer_8600 = ADR(%ID296); AdrOffset_8600 = 4294967295; BitOffset_8600 = 0; BitLength_8600 = 0; Address_8610 = ''; Type_8610 = ''; AddressPointer_8610 = 0; AdrOffset_8620 = 1172; BitOffset_8620 = 0; BitLength_8620 = 32; Address_8620 = '%ID293'; Type_8620 = 'DINT'; AddressPointer_8620 = ADR(%ID293)
      S02_PPU_Module : CL3-EC808AC(COE), Leadshine Technology Co.,Ltd., order no. CL3-EC808AC, version Revision=16#00000001
          settings: AutoUpdate = False; DC sync0 cycletime = 8000; DC sync1 cycletime = 8000; Number of SDO = 5; Homing Velocity (fast).Index = 16#6099; Homing Velocity (fast).Subindex = 16#01; Homing Velocity (fast).Value = 2000; Homing Velocity (fast).Size = 32; Homing Velocity (fast).AbortIfError = FALSE; Homing Velocity (fast).JumpToLine = FALSE; Homing Velocity (fast).Line = 0; Homing Velocity (fast).CompleteAccess = False; Homing Acceleration.Index = 16#609A; Homing Acceleration.Subindex = 16#00; Homing Acceleration.Value = 5000; Homing Acceleration.Size = 32; Homing Acceleration.AbortIfError = FALSE; Homing Acceleration.JumpToLine = FALSE; Homing Acceleration.Line = 0; Homing Acceleration.CompleteAccess = False; Homing Velocity (slow).Index = 16#6099; Homing Velocity (slow).Subindex = 16#02; Homing Velocity (slow).Value = 100; Homing Velocity (slow).Size = 32; Homing Velocity (slow).AbortIfError = FALSE; Homing Velocity (slow).JumpToLine = FALSE; Homing Velocity (slow).Line = 0; Homing Velocity (slow).CompleteAccess = False; Homing Method.Index = 16#6098; Homing Method.Subindex = 16#00; Homing Method.Value = 27; Homing Method.Size = 8; Homing Method.AbortIfError = FALSE; Homing Method.JumpToLine = FALSE; Homing Method.Line = 0; Homing Method.CompleteAccess = False; Modes of Operation.Index = 16#6060; Modes of Operation.Subindex = 16#00; Modes of Operation.Value = 8; Modes of Operation.Size = 8;
            Modes of Operation.AbortIfError = FALSE; Modes of Operation.JumpToLine = FALSE; Modes of Operation.Line = 0; Modes of Operation.CompleteAccess = False
          unmapped channels: Control Word, Profile Target Position, Touch Probe Function, Last Error Code, Status Word, Modes of Operation display, Position Actual Value, Touch Probe Status, Touch Probe 1 Positive Value, Digital Inputs
        Axis_5 : Axis, 3S - Smart Software Solutions GmbH, order no. 0, version 4.0.0.0
            settings: wDriveID = 4; dwRatioTechUnitsDenom = 8192; iRatioTechUnitsNum = 45; ScalingIncs = 16#10000; ScalingUnits = 360; AdrOffset_8010 = 1024; BitOffset_8010 = 0; BitLength_8010 = 16; Address_8010 = '%QW512'; Type_8010 = 'UINT'; AddressPointer_8010 = ADR(%QW512); AdrOffset_8020 = 1028; BitOffset_8020 = 0; BitLength_8020 = 32; Address_8020 = '%QD257'; Type_8020 = 'DINT'; AddressPointer_8020 = ADR(%QD257); AdrOffset_8030 = 4294967295; BitOffset_8030 = 0; BitLength_8030 = 0; Address_8030 = ''; Type_8030 = ''; AddressPointer_8030 = 0; AdrOffset_8040 = 4294967295; BitOffset_8040 = 0; BitLength_8040 = 0; Address_8040 = ''; Type_8040 = ''; AddressPointer_8040 = 0; AdrOffset_8050 = 4294967295; BitOffset_8050 = 0; BitLength_8050 = 0; Address_8050 = ''; Type_8050 = ''; AddressPointer_8050 = 0; AdrOffset_8060 = 1032; BitOffset_8060 = 0; BitLength_8060 = 16; Address_8060 = '%QW516'; Type_8060 = 'UINT';
              AddressPointer_8060 = ADR(%QW516); AdrOffset_8070 = 4294967295; BitOffset_8070 = 0; BitLength_8070 = 0; Address_8070 = ''; Type_8070 = ''; AddressPointer_8070 = 0; AdrOffset_8080 = 4294967295; BitOffset_8080 = 0; BitLength_8080 = 0; Address_8080 = ''; Type_8080 = ''; AddressPointer_8080 = 0; AdrOffset_8090 = 4294967295; BitOffset_8090 = 0; BitLength_8090 = 0; Address_8090 = ''; Type_8090 = ''; AddressPointer_8090 = 0; AdrOffset_8510 = 1038; BitOffset_8510 = 0; BitLength_8510 = 16; Address_8510 = '%IW519'; Type_8510 = 'UINT'; AddressPointer_8510 = ADR(%IW519); AdrOffset_8520 = 1044; BitOffset_8520 = 0; BitLength_8520 = 32; Address_8520 = '%ID261'; Type_8520 = 'DINT'; AddressPointer_8520 = ADR(%ID261); AdrOffset_8530 = 4294967295; BitOffset_8530 = 0; BitLength_8530 = 0; Address_8530 = ''; Type_8530 = ''; AddressPointer_8530 = 0; AdrOffset_8540 = 4294967295; BitOffset_8540 = 0; BitLength_8540 = 0;
              Address_8540 = ''; Type_8540 = ''; AddressPointer_8540 = 0; AdrOffset_8550 = 1040; BitOffset_8550 = 0; BitLength_8550 = 8; Address_8550 = '%IB1040'; Type_8550 = 'SINT'; AddressPointer_8550 = ADR(%IB1040); AdrOffset_8560 = 1056; BitOffset_8560 = 0; BitLength_8560 = 32; Address_8560 = '%ID264'; Type_8560 = 'UDINT'; AddressPointer_8560 = ADR(%ID264); AdrOffset_8570 = 1048; BitOffset_8570 = 0; BitLength_8570 = 16; Address_8570 = '%IW524'; Type_8570 = 'UINT'; AddressPointer_8570 = ADR(%IW524); AdrOffset_8580 = 1052; BitOffset_8580 = 0; BitLength_8580 = 32; Address_8580 = '%ID263'; Type_8580 = 'DINT'; AddressPointer_8580 = ADR(%ID263); AdrOffset_8590 = 4294967295; BitOffset_8590 = 0; BitLength_8590 = 0; Address_8590 = ''; Type_8590 = ''; AddressPointer_8590 = 0; AdrOffset_8600 = 4294967295; BitOffset_8600 = 0; BitLength_8600 = 0; Address_8600 = ''; Type_8600 = ''; AddressPointer_8600 = 0; AdrOffset_8600 = 4294967295;
              BitOffset_8600 = 0; BitLength_8600 = 0; Address_8610 = ''; Type_8610 = ''; AddressPointer_8610 = 0; AdrOffset_8620 = 4294967295; BitOffset_8620 = 0; BitLength_8620 = 0; Address_8620 = ''; Type_8620 = ''; AddressPointer_8620 = 0
    Ethernet : Ethernet, 3S - Smart Software Solutions GmbH, version 4.0.0.0
        settings: IPAddress = [192,168,1,11]; SubnetMask = [255,255,255,0]; GatewayAddress = [0,0,0,0]; MACAddress = [16#70,16#CA,16#4D,16#00,16#1B,16#7A]; NetworkInterfaceName = 'eth0'; NetworkInterfaceName = "eth0"; SaveCommunicationSettings = FALSE
      EtherNetIPSlave : EtherNet/IP Adapter, Inovance, version 4.0.0.0
          settings: DeviceInfo.ProductName = 'Inovance PLC EIP Adapter'; Number of Assemblies = 5; Number of Connections = 4; Connection Settings.Connection Number = 0; Connection Settings.Trigger and Transport = 67305474; Connection Settings.Connection Parameters = 1147405317; Connection Settings.O->T Requested packet interval (µs) = 0; Connection Settings.O->T Size (Bytes) = 0; Connection Settings.T->O Requested packet interval (µs) = 0; Connection Settings.T->O Size (Bytes) = 0; Connection Settings.Target Config Size (Bytes) = 2; Connection Settings.Connection Path Size (Bytes) = 8; Connection Settings.Connection Number = 1; Connection Settings.Trigger and Transport = 33751042; Connection Settings.Connection Parameters = 1147405061; Connection Settings.O->T Requested packet interval (µs) = 0; Connection Settings.O->T Size (Bytes) = 0; Connection Settings.T->O Requested packet interval (µs) = 0; Connection Settings.T->O Size (Bytes) = 0; Connection Settings.Target Config Size (Bytes) = 0; Connection Settings.Connection Path Size (Bytes) = 6; Connection Settings.Connection Number = 2; Connection Settings.Trigger and Transport = 16973826; Connection Settings.Connection Parameters = 1147405061; Connection Settings.O->T Requested packet interval (µs) = 0; Connection Settings.O->T Size (Bytes) = 0; Connection Settings.T->O Requested packet interval (µs) = 0; Connection Settings.T->O Size (Bytes) = 0; Connection Settings.Target Config Size (Bytes) = 0; Connection Settings.Connection Path Size (Bytes) = 6; Connection Settings.Connection Number = 3; Connection Settings.Trigger and Transport = 67305474; Connection Settings.Connection Parameters = 1147405317; Connection Settings.O->T Requested packet interval (µs) = 0; Connection Settings.O->T Size (Bytes) = 0; Connection Settings.T->O Requested packet interval (µs) = 0; Connection Settings.T->O Size (Bytes) = 0; Connection Settings.Target Config Size (Bytes) = 0; Connection Settings.Connection Path Size (Bytes) = 6; std:ARRAY[0..7] OF BYTE = [16#20,16#04,16#24,16#78,16#2C,16#64,16#2C,16#6E];
            std:ARRAY[0..5] OF BYTE = [16#20,16#04,16#2C,16#C6,16#2C,16#6E]; std:ARRAY[0..5] OF BYTE = [16#20,16#04,16#2C,16#C7,16#2C,16#6E]; std:ARRAY[0..5] OF BYTE = [16#20,16#04,16#2C,16#64,16#2C,16#6E];  = 0
        DWORD_Input_Module : DWORD Input Module, Inovance, order no. 2, version 4.0.0.0
            settings: DeviceInfo.ProductName = 'DWord Input Module'; DeviceInfo.ProductCode = 103; ConsumingAssemblyID = 100; DWord to slave.ReadOnly = False; DWord to slave.BitSize = 32; DWord to slave.DataSize = 4; ConfigVersion = 1140850688
            unmapped channels: %ID1000 DWord to slave
        DWORD_Output_Module : DWORD Output Module, Inovance, order no. 7, version 4.0.0.0
            settings: DeviceInfo.ProductName = 'DWord Output Module'; DeviceInfo.ProductCode = 107; ProducingAssemblyID = 110; DWord to master.ReadOnly = False; DWord to master.BitSize = 32; DWord to master.DataSize = 4; ConfigVersion = 1140850688
            unmapped channels: %QD1000 DWord to master
  SMElement/
    SM8704_SM9215
    SM4096_SM4607
    SM3584_SM4095
    SM6656_SM7167
    SM6144_SM6655
    SM0_SM511
    SM7168_SM7679
    SM8192_SM8703
    SM5120_SM5631
    SM9216_SM9727
    SM1536_SM2047
    SM9728_SM9999
    SM4608_SM5119
    SM512_SM1023
    SM7680_SM8191
    SM5632_SM6143
    SM1024_SM1535
    SM2560_SM3071
    SM3072_SM3583
    SM2048_SM2559
  SDElement/
    SD1024_SD1535
    SD6656_SD7167
    SD1536_SD2047
    SD4096_SD4607
    SD3072_SD3583
    SD6144_SD6655
    SD0_SD511
    SD5632_SD6143
    SD8192_SD8703
    SD2560_SD3071
    SD5120_SD5631
    SD2048_SD2559
    SD8704_SD9215
    SD7680_SD8191
    SD4608_SD5119
    SD9728_SD9999
    SD3584_SD4095
    SD9216_SD9727
    SD512_SD1023
    SD7168_SD7679
*)

// Device/Application/DUTS/IO/EC6_0032A
TYPE EC6_0032A :
STRUCT
	OUTPUT          :DWORD;
END_STRUCT
END_TYPE

// Device/Application/FB/11_AxisFB/DUTs/ST_DataAxis
TYPE ST_DataAxis :
STRUCT
	rJogVelocity				: REAL:= 10;			//Jog速度
	rManualVelocity			: REAL:= 50;			//手动速度
	rAutoVelocity				: REAL:= 100;			//自动速度
	rJogAcceleration    : REAL:= 50;      //轴Jog加速度
	rJogDeceleration    : REAL:= 50;      //轴Jog减速度
	rVelocityAcc        : REAL:= 50;      //连续运行加速度
	rVelocityDec        : REAL:= 50;      //连续运行减速度
	rMoveAcceleration   : REAL:= 50;      //轴定位加速度                   	
	rMoveDeceleration   : REAL:= 50;      //轴定位减速度  
	rMovePosition				: ARRAY[0..gc_uiAxisMoveNum] OF REAL;//绝对定位位置
	rMoveVelocity				: ARRAY[0..gc_uiAxisMoveNum] OF REAL;//绝对定位速度
	rRelativeDistance   : REAL;         //相对定位距离
	rRelativeVelocity   : REAL;         //相对定位速度
	rVelocityVel        : REAL;         //连续运行速度
	tMoveInPos					: ARRAY[1..gc_uiAxisMoveNum] OF TIME:=[gc_uiAxisMoveNum(T#0.1S)];//绝对定位到位延时
	rModuloHome					: REAL;					//模长内定位初始角度
	tModuloInPos				: TIME;					//模长内定位到位延时
END_STRUCT
END_TYPE

// Device/Application/DUTS/Machine/ST_CardtSta
TYPE ST_CardtSta :
STRUCT
	Card_OK             :BOOL;    //放卡完成 
	A                   :BOOL;    //A有料
	B                   :BOOL;    //B有料
	Desiccant_OK        :BOOL;    //干燥剂放料完成 
	Pushcard_OK         :BOOL;    //推卡完成
END_STRUCT
END_TYPE

// Device/Application/DUTS/HMI/ST_HMI_Vac_Pers
TYPE ST_HMI_Vac_Pers :
STRUCT
	iBreakDelay					: INT;					//破真空状态延时
	iVacuumDelay				: int;					//吸真空状态延时
	

END_STRUCT
END_TYPE

// Device/Application/DUTS/HMI/ST_HMI_Cyl_Pers
TYPE ST_HMI_Cyl_Pers :
STRUCT
	iHP_Delay					: INT;					//原点状态延时
	iWP_Delay					: INT;					//动点状态延时
END_STRUCT
END_TYPE

// Device/Application/DUTS/HMI/ST_HMI_Mac_Pers
TYPE ST_HMI_Mac_Pers :
STRUCT
	udiGoods						:  UDINT;	//当前良品数量
	udiBads				  		:  UDINT;	//当前不良数量
	udiTotal						:  UDINT;	//当前总数量 
	rYield					  	:  REAL;	//当前良品率
	rReject				  		:  REAL;	//当前不良率	
END_STRUCT
END_TYPE

// Device/Application/DUTS/IO/EC6_1616_Output
TYPE EC6_1616_Output :
STRUCT
	OUTPUT          :WORD;
END_STRUCT
END_TYPE

// Device/Application/DUTS/CT/ST_CT
TYPE ST_CT :
STRUCT
S01_Total            :REAL ;//工站节拍
S01_CY_Lifter_HP     :REAL;//升降气缸回原点时间
S01_CY_Lifter_WP     :REAL;//升降气缸回动点时间
S01_CY_Rotate_HP     :REAL;//旋转气缸回原点时间
S01_CY_Rotate_WP     :REAL;//旋转气缸回动点时间
S01_Cy_takeClamp12_HP :REAL;//夹爪12气缸回原点时间
S01_Cy_takeClamp12_WP :REAL;//夹爪12气缸回动点时间
S01_Cy_takeClamp34_HP :REAL;//夹爪34气缸回原点时间
S01_Cy_takeClamp34_WP :REAL;//夹爪34气缸回动点时间
//----------------------------------------
S02_Total            :REAL ;//工站节拍
S02_AXIS_POS1        :REAL ;//去待机位时间
S02_AXIS_POS2        :REAL ;//去放料位时间
S02_AXIS_POS3        :REAL ;//去取料位时间
//-------------------------------------------
S03_Total            :REAL;//工站节拍
S03_AXIS_Relative    :REAL;//供袋环形线移动时间
s03_CY_Lifter_HP     :REAL;//升降气缸回原点时间
s03_CY_Lifter_WP     :REAL;//升降气缸回动点时间
//----------------------------------
S04_Total            :REAL;//工站节拍
S04_Cy_push1_HP      :REAL;//推料气缸1回原点时间
S04_Cy_push1_WP      :REAL;//推料气缸1回动点时间
S04_Cy_push2_HP      :REAL;//推料气缸2回原点时间
S04_Cy_push2_WP      :REAL;//推料气缸2回动点时间
//----------------------------------------
S05_Total            :REAL ;//工站节拍
S05_AXIS_Relative    :REAL;//产品环形线移动时间
//----------------------------------
S06_Total            :REAL ;//工站节拍
S06_Cy_open_HP       :REAL;//开袋气缸回原点时间
S06_Cy_open_WP       :REAL;//开袋气缸回动点时间
S06_AXIS_POS1        :REAL ;//去取袋位时间
S06_AXIS_POS2        :REAL ;//去放袋位时间
//----------------------------------
ADD_Total            :REAL ;//工站节拍
ADD_AXIS_POS1        :REAL ;//去取料位时间
ADD_AXIS_POS2        :REAL ;//去放料位1时间
ADD_AXIS_POS3        :REAL ;//去放料位2时间
END_STRUCT
END_TYPE

// Device/Application/DUTS/Data/ST_Data
TYPE ST_Data :
STRUCT
	Axis												: ARRAY[0..gc_uiAxisNum] OF ST_DataAxis;//AXIS_FB中结构体
  Vac_Pers                    : ARRAY [0..gc_uiVacuumNum] OF ST_HMI_Vac_Pers;  //真空发生器判断延时
	Cy_Pers                     : ARRAY [0..gc_uiCylinderNum] OF ST_HMI_Cyl_Pers;//气缸到位判断延时

END_STRUCT
END_TYPE

// Device/Application/DUTS/IO/EC6_3200A
TYPE EC6_3200A :
STRUCT
	INPUT          :DWORD;
END_STRUCT
END_TYPE

// Device/Application/FB/12_BlinkFB/ST_SysPulse
TYPE ST_SysPulse :
STRUCT
	xP10ms						: BOOL;					//10ms脉冲
	xP20ms						: BOOL;					//20ms脉冲
	xP50ms						: BOOL;					//50ms脉冲
	xP100ms						: BOOL;					//100ms脉冲
	xP200ms						: BOOL;					//200ms脉冲
	xP500ms						: BOOL;					//500ms脉冲
	xP1s						  : BOOL;					//1s脉冲
	xP2s						  : BOOL;					//2s脉冲
	xP5s						  : BOOL;					//5s脉冲
	xP10s						  : BOOL;					//10s脉冲
	
	xR10ms						: BOOL;					//10ms脉冲上升沿
	xR20ms						: BOOL;					//20ms脉冲上升沿
	xR50ms						: BOOL;					//50ms脉冲上升沿
	xR100ms						: BOOL;					//100ms脉冲上升沿
	xR200ms						: BOOL;					//200ms脉冲上升沿
	xR500ms						: BOOL;					//500ms脉冲上升沿
	xR1s						: BOOL;					//1s脉冲上升沿
	xR2s						: BOOL;					//2s脉冲上升沿
	xR5s						: BOOL;					//5s脉冲上升沿
	xR10s						: BOOL;					//10s脉冲上升沿
	
	xF10ms						: BOOL;					//10ms脉冲下降沿
	xF20ms						: BOOL;					//20ms脉冲下降沿
	xF50ms						: BOOL;					//50ms脉冲下降沿
	xF100ms						: BOOL;					//100ms脉冲下降沿
	xF200ms						: BOOL;					//200ms脉冲下降沿
	xF500ms						: BOOL;					//500ms脉冲下降沿
	xF1s						: BOOL;					//1s脉冲下降沿
	xF2s						: BOOL;					//2s脉冲下降沿
	xF5s						: BOOL;					//5s脉冲下降沿
	xF10s						: BOOL;					//10s脉冲下降沿
END_STRUCT
END_TYPE

// Device/Application/FB/14_MachineFB/ST_OpeButton
TYPE ST_OpeButton :
STRUCT
	xStart						: BOOL;					//启动按钮
	xStop						: BOOL;					//停止按钮
	xReset						: BOOL;					//复位按钮
	xPause						: BOOL;					//暂停按钮
	xInit						: BOOL;					//初始化按钮
	xManualMode					: BOOL;					//手动模式
	xAutoMode					: BOOL;					//自动模式



END_STRUCT
END_TYPE

// Device/Application/DUTS/AXIS/ST_Ethercat
TYPE ST_Ethercat :
STRUCT
	xProRunStatus    :BOOL;//程序运行状态
	xFirstCycle		:BOOL;//上电第一周期
	xEtherCAT_OK    :BOOL;//总线状态 
END_STRUCT
END_TYPE

// Device/Application/DUTS/IO/EC6_1616_Input
TYPE EC6_1616_Input :
STRUCT
	INPUT          :word;
END_STRUCT
END_TYPE

// Device/Application/FB/14_MachineFB/ST_DataMachine
TYPE ST_DataMachine :
STRUCT
	bDummyDisabled				: BOOL;					//点检屏蔽
	nSampleSet					: UINT;					//取样数量设置
	rMasterSpeed                : REAL;                 //主轴送料速度mm/s
	rCycleTime					: REAL;					//循环时间，单位s
	nGoods						: UDINT;				//当前良品数量
	nBads						: UDINT;				//当前不良数量
	nTotal						: UDINT;				//当前总数量
	rYield						: REAL;					//当前良品率
	rReject						: REAL;					//当前不良率
	nTotalGoods					: UDINT;				//历史良品数量
	nTotalBads					: UDINT;				//历史不良数量
	nTotalOutputs				: UDINT;				//历史总数量
	rTotalYield					: REAL;					//历史良品率
	rTotalReject				: REAL;					//历史不良率
	nRunningTimer				: UDINT;				//运行时间计时器，单位100ns，除以10000单位ms
	nRunningTime				: UDINT;				//运行时间总秒数
	nRunningDays				: UDINT;				//运行时间-天
	nRunningHour				: UINT;					//运行时间-时
	nRunningMinute				: UINT;					//运行时间-分
	nRunningSecond				: UINT;					//运行时间-秒
END_STRUCT
END_TYPE

// Device/Application/DUTS/Machine/ST_Machine
TYPE ST_Machine :
STRUCT
//输入
xStartButton                    : BOOL ; //启动按钮
xStopButton                     : BOOL ; //停止 or 暂停
xResetButton                    : BOOL ; //复位按钮
xInitButton                     : BOOL ; //初始化按钮
xManualMode                     : BOOL ; //手动模式旋钮
xAutoMode                       : BOOL ; //自动模式旋钮
xEstopButton                    : ARRAY [1..2]  OF BOOL ; //急停1
xSafeDoor                       : ARRAY [1..16] OF BOOL ; //安全门
xAiron                          : BOOL; //气源
//输出
xTriLightRed                    : BOOL ;  //三色的红
xTriLightYellow                 : BOOL ;  //三色的黄
xTriLightGreen                  : BOOL ;  //三色的绿
xBuzzer                         : BOOL ;  //蜂鸣器
xStartLight                     : BOOL ;  //启动按钮灯
xStopLight                      : BOOL ;  //暂停 or 停止 按钮灯
xResetLight                     : BOOL ;  //复位按钮灯
xInitLight                      : BOOL ;  //初始化按钮灯
xLight                          : BOOL ;  //日光灯




END_STRUCT
END_TYPE

// Device/Application/DUTS/HMI/ST_HMI_Other
TYPE ST_HMI_Other :
STRUCT
		xOutCountZero                       :BOOL;
		xShieldSafetyDoor                   :BOOL;//安全门屏蔽
		xShieldBuzzer                       :BOOL;//蜂鸣器屏蔽
END_STRUCT
END_TYPE

// Device/Application/FB/05_StationFB/E_State

{attribute 'strict'}
TYPE E_State :
(
	NotReady:=0,				//未准备好
	iRunning:=1,					//运行中
	Alarm:=2,					//报警中
	Ready:=3,					//准备好
	Done:=4          //工站完成
	
)UINT;
END_TYPE

// Device/Application/DUTS/HMI/ST_HMI_PrgVer
TYPE ST_HMI_PrgVer :
STRUCT
	H_iVerson			 :STRING;//程序版本号
	H_iday               :UINT;
	H_imonth             :UINT;
	H_iyear              :UINT;
END_STRUCT
END_TYPE

// Device/Application/DUTS/AXIS/Axis_POS
{attribute 'qualified_only'}
{attribute 'strict'}
TYPE Axis_POS :
(
	enum_member := 0,
	TakePos,
	PutPos_1,
	PutPos_2
);
END_TYPE

// Device/Application/DUTS/Machine/ST_BagSta
TYPE ST_BagSta :
STRUCT
		Takebag_OK    :BOOL;    //取袋完成
		Suck_OK       :BOOL;    //吸袋完成
		Openbag_OK    :BOOL;    //开袋完成
		Loose_OK      :BOOL;    //松袋完成
END_STRUCT
END_TYPE

// Device/Application/FB/11_AxisFB/DUTs/ST_Axis_REF
TYPE ST_Axis_REF :
STRUCT
	Axis:				POINTER TO AXIS_REF_ETC_DS402_CS;
	Server:				POINTER TO ETCSlave;
END_STRUCT
END_TYPE

// Device/Application/GVLS/GVL_Standard


//掉电保持
VAR_GLOBAL PERSISTENT RETAIN
	stData                 AT %MB300000 : ST_Data;                                       //参数设置
	MachinePers            AT %MB320000 : ARRAY [0..gc_uiMachineNum] OF ST_HMI_Mac_Pers; //设备生产信息（进出料）
	ProVer 			           AT %MB331000 : ST_HMI_PrgVer;                                 //版本号管理
	
END_VAR

VAR_GLOBAL
	//轴映射变量
	RealAxis				            				: ARRAY[0..gc_uiAxisNum] 						OF ST_Axis_REF;
	//FB调用
	fbAxis	               							: ARRAY[0..gc_uiAxisNum] 						OF FB_Axis;          //轴
	fbCylinder	           							: ARRAY[0..gc_uiCylinderNum] 				OF FB_Cylinder;      //气缸
  fbVacuum			                  		: ARRAY[0..gc_uiVacuumNum]			    OF FB_Vacuum;        //真空发生器    
	fbProface		       									: ARRAY[0..gc_uiHMI_Num] 						OF FB_Proface;       //HMI
	fbMachine	           								: ARRAY[0..gc_uiMachineNum] 				OF FB_Machine;       //设备状态
	fbStation	           								: ARRAY[0..gc_uiStationNum] 				OF FB_Station;       //工站状态
	fbStCycleTime												: ARRAY[0..gc_uiStationNum]         OF FB_CycleTime;     //CT
	//EC总线状态
	EthercatStatus   			              : ST_Ethercat;                                           //EC状态
  //触摸屏额外功能
  HMI_Other                           : ST_HMI_Other; 
  //调速电机      
  Motion_cv_run                   : ARRAY [0..3] OF BOOL; //调速电机:1--前面三轨传送   2---后面四轨传送
	//振动盘运行和吹气
  Box_run                             : ARRAY [0..1] OF BOOL;//启动    
  Box_blow                            : ARRAY [0..2] OF BOOL;//吹气
     
END_VAR

// Device/Application/GVLS/GVL_IO
VAR_GLOBAL
	
//关联物理地址
//----------------本地输入输出-----------------
	alocalInput   AT %IB2 :ARRAY[1..4] OF EC6_3200A;    
	alocalOutput  AT %QB1 :ARRAY[1..3] OF EC6_0032A; 

//----------------远程输入输出---


//机台信号
	Machine_IO                  : ST_Machine;//设备IO

  xInput_local            :ARRAY[0..4,0..31] OF BOOL; 
  xOutput_local           :ARRAY[0..3,0..31] OF BOOL; 
END_VAR

// Device/Application/GVLS/GVL_Inside
VAR_GLOBAL
			
  stSysPulse         : ST_SysPulse ; //闪烁脉冲
	K                  :INT;//索引
	K1                 :INT;//索引
	j                  :INT ;
	CardState  , zero_card       :ARRAY[0..9] OF ST_CardtSta ; 
	BagState  , zero_bag         :ARRAY[0..9] OF ST_BagSta ; 
	xTryRun_ON                   :ARRAY[0..9] OF BOOL ; //空跑信号模拟
	Axis_main_ready             :BOOL;//主环形线轴ready
	xCycle_card_on              :BOOL;//试剂卡环形线上有料
	xCycle_bag_on               :BOOL;//试剂卡环形线上有料
  ct_show                     : ST_CT ;
	S03_CycleLineMoveCount      : INT;	     //试剂袋环型线移动计数
	S05_CycleLineMoveCount      : INT;	     //试剂卡环型线移动计数
	Eip_Upinput               AT %ID1000  : DWORD; //EIP 从上游输入
	Eip_Upoutput              AT %QD1000  : DWORD; //EIP 输出给上游
END_VAR

VAR_GLOBAL   CONSTANT  //声明常量，不允许在线修改
	P_on                              : BOOL :=TRUE;
	p_off                             : BOOL :=FALSE;
	Pi	                              : LREAL:=3.14159265358979323846264338327950238;
	gc_xEstopYesORno                  : BOOL :=0;//机器拍急停:1-停机重新初始化，0-继续跑不用初始化
	gc_uiAxisNum					  					: INT  :=5;//轴数量
	gc_uiAxisMoveNum                  : INT  :=4 ;//轴点位数量
	gc_uiCylinderNum				  				: INT  :=24;//气缸数量 (双控)
	gc_uiVacuumNum					          : INT  :=6;//真空发生器数量
  gc_uiStationNum				      			: INT  :=7;//工站数量
	gc_uiHMI_Num					  					: INT  :=2;//人机界面数量
	gc_uiMachineNum				      			: INT  :=1;//机器数量
  gc_S01CycleLineMoveCount 			    : INT  :=2;//SO1环形线工装相对原点移动节距数,总长2200  单节距100 电机一圈200mm
	gc_S03CycleLineMoveCount 			    : INT  :=2;//S03环形线工装相对原点移动节距数,总长1800  单节距100 电机一圈200mm
	gc_rCycleLineSpacing              : INT  :=200;//环形线节距 
	gc_VacNgLimit                     : INT  :=2;  //真空NG次数设置
END_VAR

// Device/Application/PersistentVars
{attribute 'qualified_only'}
VAR_GLOBAL PERSISTENT RETAIN
END_VAR

// Device/Application/POUS/Main
PROGRAM Main
VAR
END_VAR

WLTLink();

INPUT();
Add_distributor();
S01_transplant();
S02_bowlFeeder();
S03_takebag();
S04_PushCard();
S05_CircleLine();
S06_OpenBag();
OUTPUT();
CallStandard();
ControlMachine();

END_PROGRAM

// Device/Application/POUS/01_LINK/WLTLink
PROGRAM WLTLink
VAR
	i,j  :INT;
END_VAR

FOR i:=1 TO 4 BY 1 DO
		FOR j:=0 TO 31 BY 1 DO
			IF i<=3 THEN
					xOutput_local[i,j]:=GETBIT32(alocalOutput[i].OUTPUT,j);
			END_IF
			IF i<=4 THEN
					xInput_local[i,j]:=GETBIT32(alocalInput[i].INPUT,j);
				END_IF
		END_FOR
END_FOR

END_PROGRAM

// Device/Application/POUS/01_LINK/OUTPUT
PROGRAM OUTPUT
VAR
END_VAR

//-----------------------------------模块一-----------------------------------------------
  alocalOutput[1].OUTPUT.0   :=Machine_IO.xStartLight;
  alocalOutput[1].OUTPUT.1   :=Machine_IO.xStopLight;
  alocalOutput[1].OUTPUT.2   :=Machine_IO.xResetLight;
  alocalOutput[1].OUTPUT.3   :=Machine_IO.xInitLight;
//alocalOutput[1].OUTPUT.4   :=
  alocalOutput[1].OUTPUT.5   :=Machine_IO.xTriLightYellow  := fbMachine[1].xLampYellow; 
  alocalOutput[1].OUTPUT.6   :=Machine_IO.xTriLightGreen   := fbMachine[1].xLampGreen;
  alocalOutput[1].OUTPUT.7   :=Machine_IO.xTriLightRed     :=fbMachine[1].xLampRed;  
  alocalOutput[1].OUTPUT.8   :=Machine_IO.xBuzzer          := fbMachine[1].xLampBuzzer;
//alocalOutput[1].OUTPUT.9   :=Add_distributor.Cy_takeClamp1_1.xHP_Valve;
  alocalOutput[1].OUTPUT.10  :=Add_distributor.Cy_takeClamp1_1.xWP_Valve; //分料夹爪气缸一拖6
 (* alocalOutput[1].OUTPUT.11  :=Add_distributor.Cy_takeClamp1_2.xHP_Valve;
  alocalOutput[1].OUTPUT.12  :=Add_distributor.Cy_takeClamp1_2.xWP_Valve;
  alocalOutput[1].OUTPUT.13  :=Add_distributor.Cy_takeClamp2_1.xHP_Valve;
  alocalOutput[1].OUTPUT.14  :=Add_distributor.Cy_takeClamp2_1.xWP_Valve;
  alocalOutput[1].OUTPUT.15  :=Add_distributor.Cy_takeClamp2_2.xHP_Valve;
  alocalOutput[1].OUTPUT.16  :=Add_distributor.Cy_takeClamp2_2.xWP_Valve;
  alocalOutput[1].OUTPUT.17  :=Add_distributor.Cy_takeClamp3_1.xHP_Valve;
  alocalOutput[1].OUTPUT.18  :=Add_distributor.Cy_takeClamp3_1.xWP_Valve;
  alocalOutput[1].OUTPUT.19  :=Add_distributor.Cy_takeClamp3_2.xHP_Valve;
  alocalOutput[1].OUTPUT.20  :=Add_distributor.Cy_takeClamp3_2.xWP_Valve;*)
//alocalOutput[1].OUTPUT.21  :=Add_distributor.Cy_openleft.xHP_Valve;
  alocalOutput[1].OUTPUT.22  :=Add_distributor.Cy_openleft.xWP_Valve;//单控阀
//alocalOutput[1].OUTPUT.23  :=Add_distributor.Cy_openright.xHP_Valve;
  alocalOutput[1].OUTPUT.24  :=Add_distributor.Cy_openright.xWP_Valve;//单控阀
  alocalOutput[1].OUTPUT.25  :=Add_distributor.Cy_lifter.xHP_Valve;
  alocalOutput[1].OUTPUT.26  :=Add_distributor.Cy_lifter.xWP_Valve;
//alocalOutput[1].OUTPUT.27  :=
//alocalOutput[1].OUTPUT.28  :=
//alocalOutput[1].OUTPUT.29  :=
//alocalOutput[1].OUTPUT.30  :=
//alocalOutput[1].OUTPUT.31  :=

//-----------------------------------模块二-----------------------------------------------
//alocalOutput[2].OUTPUT.0  :=S01_transplant.Cy_rotate.xHP_Valve;
  alocalOutput[2].OUTPUT.1  :=S01_transplant.Cy_rotate.xWP_Valve;        //单控阀
//alocalOutput[2].OUTPUT.2  :=S01_transplant.Cy_takeClamp1.xHP_Valve;
  alocalOutput[2].OUTPUT.3  :=S01_transplant.Cy_takeClamp1.xWP_Valve;    //单控阀
//alocalOutput[2].OUTPUT.4  :=S01_transplant.Cy_takeClamp2.xHP_Valve;
//alocalOutput[2].OUTPUT.5  :=S01_transplant.Cy_takeClamp2.xWP_Valve;
//alocalOutput[2].OUTPUT.6  :=S01_transplant.Cy_takeClamp3.xHP_Valve;
  alocalOutput[2].OUTPUT.7  :=S01_transplant.Cy_takeClamp3.xWP_Valve;    //单控阀
//alocalOutput[2].OUTPUT.8  :=S01_transplant.Cy_takeClamp4.xHP_Valve;
//alocalOutput[2].OUTPUT.9  :=S01_transplant.Cy_takeClamp4.xWP_Valve;
  alocalOutput[2].OUTPUT.10 :=S01_transplant.Cy_lifter.xHP_Valve;
  alocalOutput[2].OUTPUT.11 :=S01_transplant.Cy_lifter.xWP_Valve;
//alocalOutput[2].OUTPUT.12 :=
//alocalOutput[2].OUTPUT.13 :=
//alocalOutput[2].OUTPUT.14 :=
//alocalOutput[2].OUTPUT.15 :=
  alocalOutput[2].OUTPUT.16 :=S02_bowlFeeder.Cy_resist_1.xHP_Valve;
  alocalOutput[2].OUTPUT.17 :=S02_bowlFeeder.Cy_resist_1.xWP_Valve;
  alocalOutput[2].OUTPUT.18 :=S02_bowlFeeder.Cy_resist_2.xHP_Valve;
  alocalOutput[2].OUTPUT.19 :=S02_bowlFeeder.Cy_resist_2.xWP_Valve;
  alocalOutput[2].OUTPUT.20 :=S02_bowlFeeder.Cy_resist_3.xHP_Valve;
  alocalOutput[2].OUTPUT.21 :=S02_bowlFeeder.Cy_resist_3.xWP_Valve;
  alocalOutput[2].OUTPUT.22 :=S02_bowlFeeder.Cy_resist_4.xHP_Valve;
  alocalOutput[2].OUTPUT.23 :=S02_bowlFeeder.Cy_resist_4.xWP_Valve;
  alocalOutput[2].OUTPUT.24 :=Motion_cv_run[1];
  alocalOutput[2].OUTPUT.25 :=Motion_cv_run[2];
  alocalOutput[2].OUTPUT.26 :=Motion_cv_run[3];
  alocalOutput[2].OUTPUT.27 :=Machine_IO.xLight  ;//日光灯
//alocalOutput[2].OUTPUT.28 :=
//alocalOutput[2].OUTPUT.29 :=
//alocalOutput[2].OUTPUT.30 :=
//alocalOutput[2].OUTPUT.31 :=

//-----------------------------------模块三-----------------------------------------------
  alocalOutput[3].OUTPUT.0   :=S02_bowlFeeder.Va_ppu_1.xVacuumValve;
  alocalOutput[3].OUTPUT.1   :=S02_bowlFeeder.Va_ppu_1.xBreakValve;
  alocalOutput[3].OUTPUT.2   :=S02_bowlFeeder.Va_ppu_2.xVacuumValve;
  alocalOutput[3].OUTPUT.3   :=S02_bowlFeeder.Va_ppu_2.xBreakValve;
  alocalOutput[3].OUTPUT.4   :=S03_takebag.Cy_BinLifter.xHP_Valve;
  alocalOutput[3].OUTPUT.5   :=S03_takebag.Cy_BinLifter.xWP_Valve;
//alocalOutput[3].OUTPUT.6   :=
//alocalOutput[3].OUTPUT.7   :=
//alocalOutput[3].OUTPUT.8   :=S03_takebag.Cy_lifter.xHP_Valve;
  alocalOutput[3].OUTPUT.9   :=S03_takebag.Cy_lifter.xWP_Valve;
  alocalOutput[3].OUTPUT.10  :=S03_takebag.Va_take1.xVacuumValve;
//alocalOutput[3].OUTPUT.11  :=S03_takebag.Va_take1.xBreakValve;
  alocalOutput[3].OUTPUT.12  :=S03_takebag.Va_take2.xVacuumValve;
//alocalOutput[3].OUTPUT.13  :=S03_takebag.Va_take2.xBreakValve;
//alocalOutput[3].OUTPUT.14  :=S06_packcard.Cy_open.xHP_Valve;
  alocalOutput[3].OUTPUT.15  :=S06_OpenBag.Cy_open.xWP_Valve;
  alocalOutput[3].OUTPUT.16  :=S06_OpenBag.Va_open_left.xVacuumValve;
//alocalOutput[3].OUTPUT.17  :=S06_packcard.Va_open_left.xBreakValve;
  alocalOutput[3].OUTPUT.18  :=S06_OpenBag.Va_open_right.xVacuumValve;
//alocalOutput[3].OUTPUT.19  :=S06_packcard.Va_open_right.xBreakValve;
  alocalOutput[3].OUTPUT.20  :=Box_blow[1];
  alocalOutput[3].OUTPUT.21  :=Box_blow[2];
  alocalOutput[3].OUTPUT.22  :=Box_run[1];
//alocalOutput[3].OUTPUT.23  :=
  alocalOutput[3].OUTPUT.24  :=S03_takebag.Cy_BinInsert.xHP_Valve;
  alocalOutput[3].OUTPUT.25  :=S03_takebag.Cy_BinInsert.xWP_Valve;
//alocalOutput[3].OUTPUT.26  :=S04_bagging.Cy_push1.xHP_Valve;
  alocalOutput[3].OUTPUT.27 :=S04_PushCard.Cy_push1.xWP_Valve;
//alocalOutput[3].OUTPUT.28  :=S04_bagging.Cy_push2.xHP_Valve;
  alocalOutput[3].OUTPUT.29 :=S04_PushCard.Cy_push2.xWP_Valve;
//alocalOutput[3].OUTPUT.30  :=
//alocalOutput[3].OUTPUT.31  :=

END_PROGRAM

// Device/Application/POUS/02_STATION/Add_distributor
PROGRAM Add_distributor
VAR_INPUT
	//工站
	station					    : REFERENCE TO FB_Station:=fbStation[7];//工站状态
	cycleTime						: REFERENCE TO FB_CycleTime:= fbStCycleTime[7];	//工站CT
//伺服
	Axis_distributor	  : REFERENCE TO FB_Axis:=fbAxis[5];
//气缸
	Cy_takeClamp1_1				    : REFERENCE TO FB_Cylinder:=fbCylinder[16];//1轨前夹爪
	//Cy_takeClamp1_2				    : REFERENCE TO FB_Cylinder:=fbCylinder[17];//1轨后夹爪
	//Cy_takeClamp2_1				    : REFERENCE TO FB_Cylinder:=fbCylinder[18];//2轨前夹爪
	//Cy_takeClamp2_2				    : REFERENCE TO FB_Cylinder:=fbCylinder[19];//2轨后夹爪
	//Cy_takeClamp3_1				    : REFERENCE TO FB_Cylinder:=fbCylinder[20];//3轨前夹爪
  //Cy_takeClamp3_2				    : REFERENCE TO FB_Cylinder:=fbCylinder[21];//3轨后夹爪
	Cy_openleft			          : REFERENCE TO FB_Cylinder:=fbCylinder[22];//左开气缸
  Cy_openright			        : REFERENCE TO FB_Cylinder:=fbCylinder[23];//右开气缸
  Cy_lifter			            : REFERENCE TO FB_Cylinder:=fbCylinder[24];//升降气缸
	//传感器
	Sensor_cvfront_on        : ARRAY[0..6] OF BOOL; //三轨到位传感器
	Sensor_cvback_on            : ARRAY[0..4] OF BOOL; //四轨满料传感器
	//调速电机
	
	
END_VAR

VAR
		arTon               :ARRAY[0..10] OF ton ; 
		arTon_alarm         :ARRAY[0..10] OF ton ; 
		xCV_take_full       :BOOL; //三轨满料
		xCV_put_full        :BOOL; //四轨有料
    xPut_mark           :BOOL; //放料标识
    rt_Ctmark           :R_TRIG;
		i                   :INT;
		CT_DisAction        : ARRAY[0..10] OF FB_CycleTime;
		CT_DisAction_1      : ARRAY[0..10] OF FB_CycleTime_1;			
	  CT_DisAction_2      : ARRAY[0..10] OF FB_CycleTime_2;		
    Rt_Alarm            : ARRAY[0..31] OF R_TRIG;
END_VAR

Alarm();
Delay();
FlowAuto();
FlowInit();
General();
ILC();
TipAuto();
TipManual();

ACTION ILC:

//---------------------------------------------------工站可执行-------------------------------------------------------
station.xCanRun := TRUE ;

//---------------------------------------------------气缸动作条件-------------------------------------------
Cy_takeClamp1_1.xOnILC:=
Cy_takeClamp1_1.xOffILC:=TRUE;

(*Cy_takeClamp1_2.xOnILC:=
Cy_takeClamp1_2.xOffILC:=TRUE;

Cy_takeClamp2_1.xOnILC:=
Cy_takeClamp2_1.xOffILC:=TRUE;

Cy_takeClamp2_2.xOnILC:=
Cy_takeClamp2_2.xOffILC:=TRUE;

Cy_takeClamp3_1.xOnILC:=
Cy_takeClamp3_1.xOffILC:=TRUE;

Cy_takeClamp3_2.xOnILC:=
Cy_takeClamp3_2.xOffILC:=TRUE;*)

Cy_lifter.xOnILC:=
Cy_lifter.xOffILC:= TRUE;

Cy_openleft.xOnILC:=
Cy_openleft.xOffILC:= TRUE;

Cy_openright.xOnILC:=
Cy_openright.xOffILC:= TRUE;



//---------------------------------------------------伺服动作条件-------------------------------------------
Axis_distributor.xJogILC :=     
Axis_distributor.xHomeILC := 
Axis_distributor.xRunILC := 
Axis_distributor.xRelativeILC:=
Axis_distributor.xMoveILC[1] :=                            //取料位
Axis_distributor.xMoveILC[2] :=                            //放料位1
Axis_distributor.xMoveILC[3] := TRUE;                      //放料位2
END_ACTION

ACTION Alarm:
//工站初始化
station.adwAlarm[1].00:=station.xInitTimeout;	             //Add_distributor 工站初始化超时报警
//气缸
station.adwAlarm[1].01:=	Cy_takeClamp1_1.xHP_Off ;        //Add_distributor Cy_takeClamp1_1 夹爪1 气缸原点无信号
station.adwAlarm[1].02:=	Cy_takeClamp1_1.xWP_Off ;        //Add_distributor Cy_takeClamp1_1 夹爪1 气缸动点无信号
//station.adwAlarm[1].03:=	Cy_takeClamp2_1.xHP_Off ;        //
//station.adwAlarm[1].04:=	Cy_takeClamp2_1.xWP_Off ;        //
//station.adwAlarm[1].05:=	Cy_takeClamp3_1.xHP_Off ;        //
//station.adwAlarm[1].06:=	Cy_takeClamp3_1.xWP_Off ;        //
//station.adwAlarm[1].07:=	Cy_takeClamp1_2.xHP_Off ;        //
//station.adwAlarm[1].08:=	Cy_takeClamp1_2.xWP_Off;         //
//station.adwAlarm[1].09:=	Cy_takeClamp2_2.xHP_Off;         //
//station.adwAlarm[1].10:=	Cy_takeClamp2_2.xWP_Off ;        //
//station.adwAlarm[1].11:=	Cy_takeClamp3_2.xHP_Off ;        //
//station.adwAlarm[1].12:=	Cy_takeClamp3_2.xWP_Off ;        //
station.adwAlarm[1].13:=	Cy_openleft.xHP_Off ;            //
station.adwAlarm[1].14:=	Cy_openleft.xWP_Off;             //
station.adwAlarm[1].15:=	Cy_openright.xHP_Off;            //
station.adwAlarm[1].16:=	Cy_openright.xWP_Off ;           //
station.adwAlarm[1].17:=	Cy_lifter	.xHP_Off;              //
station.adwAlarm[1].18:=	Cy_lifter	.xWP_Off ;             //
//轴
station.adwAlarm[1].19:=	Axis_distributor.xError ;            //轴报错
station.adwAlarm[1].20:=	Axis_distributor.xNotPowerOn;         //未使能
station.adwAlarm[1].21:=	Axis_distributor.xMoveTimeout;        //定位超时
//流程
station.adwAlarm[1].22:=arTon_alarm[1].Q OR arTon_alarm[2].Q OR arTon_alarm[3].Q OR arTon_alarm[4].Q;//四轨满料报警
END_ACTION

ACTION Delay:

//----------------------------------------------动作延时-----------------------------------------------

arTon[1](IN:=NOT (Sensor_cvback_on[1] OR Sensor_cvback_on [2] OR Sensor_cvback_on[3] OR Sensor_cvback_on [4]) , PT:=T#100MS , Q=> , ET=> );//四轨有料判断
arTon[2](IN:= Cy_takeClamp1_1.xHP_Delay AND station.iStepAuto=30, PT:=T#500MS , Q=> , ET=> );//张开延时
arTon[3](IN:=   , PT:=T#60S , Q=> , ET=> );//

//----------------------------------------------报警延时-----------------------------------------------
arTon_alarm[1](IN:= Sensor_cvback_on[1] AND station.xRunning , PT:=T#7S , Q=> , ET=> );//轨1满料
arTon_alarm[2](IN:= Sensor_cvback_on[2] AND station.xRunning , PT:=T#7S , Q=> , ET=> );//轨2满料
arTon_alarm[3](IN:= Sensor_cvback_on[3] AND station.xRunning , PT:=T#7S , Q=> , ET=> );//轨3满料
arTon_alarm[4](IN:= Sensor_cvback_on[4] AND station.xRunning , PT:=T#7S , Q=> , ET=> );//轨4满料
arTon_alarm[5](IN:= NOT Axis_distributor.xbusy  , PT:=T#1S , Q=> , ET=> );//轴到位判断延时
arTon_alarm[6](IN:=   , PT:=T#60S , Q=> , ET=> );//

arTon_alarm[7](IN:=   , PT:=T#10S , Q=> , ET=> );//
arTon_alarm[8](IN:=   , PT:=T#60S , Q=> , ET=> );//
arTon_alarm[9](IN:=   , PT:=T#60S , Q=> , ET=> );//
END_ACTION

ACTION TipManual:
//--------------------------------------------ManualTip------------------------------------------------------
station.adwManualTip[1].00			:=FALSE;//提示1
//-------------------------------------------气缸提示---------------------------------------------------------




/////////////////////////////////////////////////////////////////////////////////////////////////////////////////
END_ACTION

ACTION TipAuto:

//------------------------------------------------AutoTip General---------------------------------


//------------------------------------------------AutoTip Cylinder--------------------------------

station.adwAutoTip[1].00:=FALSE;	//
station.adwAutoTip[1].01:=FALSE;	//
station.adwAutoTip[1].02:=Cy_takeClamp1_1.xAutoTip;	   //夹爪1 气缸自动中有手动
(*station.adwAutoTip[1].03:=Cy_takeClamp2_1.xAutoTip;	   //夹爪2 气缸自动中有手动
station.adwAutoTip[1].04:=Cy_takeClamp3_1.xAutoTip;	   //夹爪3 气缸自动中有手动
station.adwAutoTip[1].05:=Cy_takeClamp1_2.xAutoTip;	   //夹爪4 气缸自动中有手动
station.adwAutoTip[1].06:=Cy_takeClamp2_2.xAutoTip;	   //夹爪5 气缸自动中有手动
station.adwAutoTip[1].07:=Cy_takeClamp3_2.xAutoTip;	   //夹爪6 气缸自动中有手动*)
station.adwAutoTip[1].08:=Cy_openleft.xAutoTip;	       //左变距 气缸自动中有手动
station.adwAutoTip[1].09:=Cy_openright.xAutoTip;	     //右变距 气缸自动中有手动
station.adwAutoTip[1].10:=Cy_lifter	.xAutoTip;	       //升降   气缸自动中有手动
//伺服位置的读取,伺服位置错误自动提示               //Axis_distributor自动时位置错误
   FOR i:= 1 TO 5 BY 1 DO 
   	IF Axis_distributor.xMoveAuto[i] THEN
   		Axis_distributor.iPosNumber := i ;
   	END_IF
   END_FOR
IF fbMachine[1].xAutoMode AND NOT fbMachine[1].xRunning AND arTon_alarm[5].Q THEN 
	IF Axis_distributor.iPosNumber=1 AND NOT Axis_distributor.xMoveInPos[1] THEN station.adwAutoTip[1].11:=TRUE; END_IF //Axis_distributor自动时位置不在位置1
	IF Axis_distributor.iPosNumber=2 AND NOT Axis_distributor.xMoveInPos[2] THEN station.adwAutoTip[1].12:=TRUE; END_IF //Axis_distributor自动时位置不在位置2
	IF Axis_distributor.iPosNumber=3 AND NOT Axis_distributor.xMoveInPos[3] THEN station.adwAutoTip[1].13:=TRUE; END_IF //Axis_distributor自动时位置不在位置3
END_IF
END_ACTION

ACTION General:
//三轨满料判断
IF Sensor_cvfront_on[1] AND Sensor_cvfront_on [2] AND Sensor_cvfront_on[3] 
AND Sensor_cvfront_on [4] AND  Sensor_cvfront_on[5] AND Sensor_cvfront_on [6]
THEN
xCV_take_full:=TRUE;
ELSE
xCV_take_full:=FALSE;	
END_IF



//CT
rt_Ctmark(CLK:=Cy_takeClamp1_1.xAuto , Q=>cycleTime.xCycleMark );

CT_DisAction_2[1](xCycleStartMark:=Cy_takeClamp1_1.xHP_Valve ,xCycleEndMark:= Cy_takeClamp1_1.xHP_Delay,xCycleRun:=TRUE, RCycleTime=>ct_show.S01_Cy_takeClamp12_HP);
CT_DisAction_2[2](xCycleStartMark:=Cy_takeClamp1_1.xWP_Valve ,xCycleEndMark:= Cy_takeClamp1_1.xWP_Delay,xCycleRun:=TRUE, RCycleTime=>ct_show.S01_Cy_takeClamp12_WP);
CT_DisAction_2[4](xCycleStartMark:=Axis_distributor.xMoveAuto[1] ,xCycleEndMark:= Axis_distributor.xMoveInPos[1],xCycleRun:=TRUE, RCycleTime=>ct_show.ADD_AXIS_POS1);
CT_DisAction_2[5](xCycleStartMark:=Axis_distributor.xMoveAuto[2] ,xCycleEndMark:= Axis_distributor.xMoveInPos[2],xCycleRun:=TRUE, RCycleTime=>ct_show.ADD_AXIS_POS2);
CT_DisAction_2[6](xCycleStartMark:=Axis_distributor.xMoveAuto[3] ,xCycleEndMark:= Axis_distributor.xMoveInPos[3],xCycleRun:=TRUE, RCycleTime=>ct_show.ADD_AXIS_POS3);
END_ACTION

ACTION FlowAuto:

//-----------------------------------------初始化是否完成判断----------------------------------------------
IF NOT station.xInitDone 
THEN
 	station.iStepAuto:=0;
 	station.xDone:=FALSE;
ELSIF station.xRunning  //单循环关联到running
THEN
//-----------------------------------------动作步骤--------------------------------------------------------
CASE station.iStepAuto OF	  
	0: //----Home Step，等待启动----
		
		IF station.xDisabled AND station.xCanRun 	AND NOT fbMachine[1].xStopped AND NOT station.xSingleRunning 
		THEN
			station.xDone:=TRUE;//工站完成信号判断
		END_IF
		
	  IF  station.xSingleRunning OR station.xCanRun	AND NOT station.xDone AND NOT station.xDisabled	AND NOT fbMachine[1].xStopped
		THEN
			station.xCycleEnable:=TRUE;
			station.xDone:= FALSE;  
			station.iStepAuto:= 5;
		END_IF
		5://判断夹爪模组状态
		IF  Cy_lifter.xWP_Delay THEN
		  	Cy_lifter.xAuto:=FALSE;   //升降气缸回原位
		END_IF
		IF NOT  Cy_openright.XHP_Delay OR  NOT Cy_openleft.xHP_Delay THEN
		Cy_openright.xAuto:=FALSE;
		Cy_openleft.xAuto:=FALSE;
		END_IF
		IF Cy_lifter.xHP_Delay AND Cy_takeClamp1_1.xHP_Delay  AND  NOT Axis_distributor.xMoveInPos[1] THEN
			Axis_distributor.xMoveAuto[1]:=TRUE;//伺服去取料位
		END_IF
		IF Cy_takeClamp1_1.xHP_Delay  AND  Cy_lifter.xHP_Delay AND Axis_distributor.xMoveInPos[1]
		THEN   
		   station.iStepAuto :=10;
    END_IF 		
    10://等待取料
		IF (xCV_take_full OR fbmachine[1].xTryRun)  AND Cy_lifter.xHP_Delay AND Cy_takeClamp1_1.xHP_Delay THEN
			Cy_lifter.xAuto:=TRUE;
		END_IF
		IF Cy_lifter.xWP_Delay AND Cy_takeClamp1_1.xHP_Delay AND (xCV_take_full OR fbmachine[1].xTryRun) THEN
		Cy_takeClamp1_1.xAuto:=TRUE;	
	(*	Cy_takeClamp1_2.xAuto:=TRUE;
		Cy_takeClamp2_1.xAuto:=TRUE;
		Cy_takeClamp2_2.xAuto:=TRUE;
		Cy_takeClamp3_1.xAuto:=TRUE;
		Cy_takeClamp3_2.xAuto:=TRUE;			*)
		END_IF
		IF  Cy_takeClamp1_1.xWP_Delay THEN
			Cy_lifter.xAuto:=FALSE;
			station.iStepAuto :=20;
		END_IF
    20://去放料位判断
		IF Cy_lifter.xHP_Delay AND Cy_takeClamp1_1.xWP_Delay AND Axis_distributor.xMoveInPos[1] THEN
			 IF  xPut_mark   THEN
				 		station.iStepAuto :=200;//去放料位1动作
		   	ELSE
			    	station.iStepAuto :=300;//去放料位2动作	 		
	    	END_IF
	  END_IF		
		200://放料位1
		Cy_openright.xAuto:=TRUE;
		Cy_openleft.xAuto:=FALSE;		
		IF NOT Axis_distributor.xMoveInPos[2] THEN
        Axis_distributor.xMoveAuto[2]:=TRUE;//伺服去放料位1		
		END_IF
		IF Axis_distributor.xMoveInPos[2] AND Cy_openright.XWP_Delay AND Cy_openleft.xHP_Delay AND (NOT xCV_put_full OR fbmachine[1].xTryRun) THEN
		//Cy_lifter.xAuto:=TRUE;
		xPut_mark:=FALSE;
		station.iStepAuto :=30;
		END_IF
		300://放料位2
		Cy_openright.xAuto:=FALSE;
		Cy_openleft.xAuto:=TRUE;		
		IF NOT Axis_distributor.xMoveInPos[3] THEN
        Axis_distributor.xMoveAuto[3]:=TRUE;//伺服去放料位2	
		END_IF
		IF Axis_distributor.xMoveInPos[3] AND Cy_openleft.XWP_Delay AND Cy_openright.XHP_Delay AND (NOT xCV_put_full OR fbmachine[1].xTryRun) THEN
		//Cy_lifter.xAuto:=TRUE;
		xPut_mark:=TRUE;
		station.iStepAuto :=30;
		END_IF
		30://放料完成
    IF arTon[1].Q THEN
		Cy_takeClamp1_1.xAuto:=FALSE;	
    END_IF
		IF arTon[2].Q THEN//张开延时
 		station.iStepAuto :=40;
		END_IF
		40://回取料位	
		Cy_openright.xAuto:=FALSE;
		Cy_openleft.xAuto:=FALSE;
		Axis_distributor.xMoveAuto[1]:=TRUE;
		IF 		Cy_lifter.xHP_Delay AND Cy_openright.XHP_Delay AND  Cy_openleft.xHP_Delay AND Cy_takeClamp1_1.xHP_Delay AND Axis_distributor.xMoveInPos[1] THEN
				station.iStepAuto :=999;
		END_IF
		
		
		
		
		
		
		
		
	999://----Single Run Finish----
			
		station.iStepAuto :=0;
//		station.xDone:=TRUE;
		station.xSingleRunFlag:=FALSE;
		station.xCycleEnable:=FALSE;	
END_CASE

END_IF
END_ACTION

ACTION FlowInit:
IF NOT station.xIniting THEN
  station.iStepInit:=0;    
ELSE
//--------------------------------------------初始化步序----------------------------------
CASE station.iStepInit OF	
 0://  
  	IF station.xIniting THEN	
  	  station.iStepInit:=10;	
  	END_IF	
10://复位数据
   Motion_cv_run[1]:=FALSE;//传送带运行复位
   Motion_cv_run[2]:=FALSE;        
    station.iStepInit := 20 ;		
20://升降气缸原点
    Cy_lifter.xInit := TRUE ;
		IF Cy_lifter.xHP_Delay   THEN 
    station.iStepInit:=30;	
		END_IF
30://气缸回原点
    Cy_openleft.xInit := TRUE ;
		Cy_openright.xInit := TRUE ;
		Cy_takeClamp1_1.xInit:=TRUE;	
(*	Cy_takeClamp1_2.xInit:=TRUE;
		Cy_takeClamp2_1.xInit:=TRUE;
		Cy_takeClamp2_2.xInit:=TRUE;
		Cy_takeClamp3_1.xInit:=TRUE;
		Cy_takeClamp3_2.xInit:=TRUE;*)
    IF Cy_openleft.xHP_Delay AND Cy_openright.xHP_Delay 
			AND Cy_takeClamp1_1.xHP_Delay 
  (*  AND Cy_takeClamp1_2.xHP_Delay
			AND Cy_takeClamp2_1.xHP_Delay AND Cy_takeClamp2_2.xHP_Delay
			AND Cy_takeClamp3_1.xHP_Delay AND Cy_takeClamp3_2.xHP_Delay*)
THEN 
    station.iStepInit:=40;	
		END_IF
40://轴上使能
   	Axis_distributor.xPowerInit := TRUE ;
    IF 	Axis_distributor.xPowerOn THEN 
    		station.iStepInit:=60;	
		END_IF		
50://轴回原点,绝对值编码器，回过原点，不需要再回
    Axis_distributor.xHomeAuto := TRUE ;
		IF Axis_distributor.xHomeDone THEN
    Axis_distributor.xHomeAuto := FALSE ;
    		station.iStepInit:=60;	
		END_IF
60://轴去待机位
    Axis_distributor.xMoveAuto[1] := TRUE ;
		IF Axis_distributor.xMoveInPos[1] THEN 
    		station.iStepInit:=999;	
		END_IF			
999://初始化完成	
	station.iStepInit:=0;
	station.xInitDone:=TRUE;  
END_CASE
END_IF
END_ACTION

END_PROGRAM

// Device/Application/FB/05_StationFB/FB_Station
FUNCTION_BLOCK FB_Station
VAR_INPUT
	xEStop						: BOOL;					//急停
	xKey						: BOOL:=TRUE;			//钥匙开关
	xSafety						: BOOL;					//安全防护
	xManualMode					: BOOL;					//手动模式
	xReset						: BOOL;					//复位按钮	
	xMachinePause				: BOOL;					//整机暂停按钮
	xMachineReInit				: BOOL;					//整机重新初始化时，复位初始化完成
	xMachineIniting				: BOOL;					//整机初始化中
	xMachineRunning				: BOOL;					//整机自动中
	tInitTimeout				: TIME:=T#60S;			//初始化超时
	xPauseDisable        		: BOOL;            		//暂停失效标志位
	
	xInitHmi					: BOOL;					//初始化HMI
	xInitDone					: BOOL;					//初始化完成
	xDisabled					: BOOL;					//工站屏蔽
	xCycleRunHmi				: BOOL;					//连动HMI
	xJogRunHmi					: BOOL;					//寸动HMI
	xPauseHmi					: BOOL;					//暂停HMI
	xStop						: BOOL;					//其它条件要求工站停止运行
	xSingleRunFlag				: BOOL;					//单动标志
	xCycleEnable				: BOOL;					//循环开始，工站周期计时开始
	rWaitingTime				: REAL;					//周期等待时间，如待料，单位s  
	
	adwAlarm	          		: ARRAY[0..4] OF DWORD;	//报警		
	adwAutoTip					: ARRAY[0..4] OF DWORD;	//自动提示
	adwManualTip				: ARRAY[0..4] OF DWORD;	//手动提示
	
	xAlarm						: BOOL;					//报警中
	xAutoTip					: BOOL;					//自动提示中
	xManualTip					: BOOL;					//手动提示中
	xTip						: BOOL;					//提示中
	xDone						: BOOL;					//工站完成
	xCanRun						: BOOL;					//工站可动作
	iStepAuto           		: INT ;         		//自动流程步
	aSubStepAuto           		:ARRAY[1..10] OF INT ;         		//自动子流程步	
	iStepInit           		: INT ;         		//初始化流程步
	bAutoState					: BYTE ;				//工站自动流程状态机
END_VAR

VAR_OUTPUT
	xStationIniting				: BOOL;					//单工站初始化中
	xIniting					: BOOL;					//初始化中
	xInitTimeout				: BOOL;					//初始化超时
	xCycleRunning				: BOOL;					//连动中
	xJogRunning					: BOOL;					//寸动中
	xSingleRunning				: BOOL;					//单动中
	xRunning					: BOOL;					//运行中
	xDeviceRunning		: BOOL;					//第三方设备运行中
	uiState						: UINT;					//工站状态
	//tCycleTime				:TIME;
	diCycleTime 				: DINT;					//基础时间是100ms
	
	adwAlarmOut	          : ARRAY[0..4] OF DWORD;	//报警
	adwAutoTipOut					: ARRAY[0..4] OF DWORD;	//自动提示
	adwManualTipOut				: ARRAY[0..4] OF DWORD;	//手动提示
	//将字转换为bool
	xadwAlarm	          : ARRAY[0..4,0..31] OF BOOL;	//报警
	xadwAutoTip					: ARRAY[0..4,0..31] OF BOOL;	//自动提示
	xadwManualTip				: ARRAY[0..4,0..31] OF BOOL;	//手动提示
END_VAR

VAR
	{attribute 'hide'}
	ftInitHmi					: F_TRIG;				//初始化HMI上升沿
	{attribute 'hide'}
	rtMachineReInit				: R_TRIG;				//整机重新初始化上升沿
	{attribute 'hide'}
	xInitAble					: BOOL;					//初始化条件
	{attribute 'hide'}
	xRunAble					: BOOL;					//运行条件
	{attribute 'hide'}
	tonInitTimeout				: TON;					//初始化超时计时
	{attribute 'hide'}
	ftCycleRunHMI				: F_TRIG;				//连动HMI上升沿
	{attribute 'hide'}
	rtJogRunHMI					: R_TRIG;				//寸动HMI上升沿
	{attribute 'hide'}
	xPause						: BOOL;					//暂停
	{attribute 'hide'}
	lrCycleTimer					: LREAL;				//计时器，单位100ns，除于10000后单位ms
	{attribute 'hide'}
	lrWaitingTimer				: LREAL;				//等待时间计时器
	{attribute 'hide'}
	rtCycleTimeStop				: R_TRIG;				//工站周期计时停止上升沿
	
	ton_AutoTimeout				:TON;					//工站自动流程超时			//自动程序有BUG
	i : INT ;
	xFirstCycle : BOOL ;	
	rStationStart	  : R_TRIG;							//工站完成上升沿
	fStationRunning : R_TRIG;


END_VAR

ACT_General();
ACT_Init();
ACT_Run();
ACT_State();
ACT_CycleTime();

ACTION ACT_Init:
//	初始化条件
xInitAble:=xEStop
	AND xKey
	AND xSafety
	AND xManualMode
	AND NOT xAlarm
	AND NOT xInitTimeout;

//	急停或初始化时先复位初始化完成
ftInitHmi(CLK:=xInitHmi, Q=>);
rtMachineReInit(CLK:=xMachineReInit, Q=>);

IF ((NOT xEStop OR rtMachineReInit.Q OR ftInitHmi.Q )AND gc_xEstopYesORno)OR 
	 (( rtMachineReInit.Q OR ftInitHmi.Q AND xInitAble)AND NOT gc_xEstopYesORno)
THEN
	xInitDone:=FALSE;
END_IF

//	单工站初始化中
IF xInitAble
	AND NOT xInitDone
	AND NOT xInitTimeout
	AND NOT xPause
	AND NOT xMachineIniting
THEN
	IF ftInitHmi.Q THEN
		xStationIniting:=TRUE;
	END_IF
ELSE
	xStationIniting:=FALSE;
END_IF

//	初始化中
xIniting:=xStationIniting
	OR xMachineIniting
		AND xInitAble
		AND NOT xInitDone;

//	初始化超时
tonInitTimeout(
	IN:=xIniting,
	PT:=tInitTimeout,
	Q=>, ET=>);
IF xReset THEN
	xInitTimeout:=FALSE;
END_IF
IF tonInitTimeout.Q THEN
	xInitTimeout:=TRUE;
END_IF
END_ACTION

ACTION ACT_State:


//	未准备好
IF NOT xInitDone
	AND NOT xAlarm
THEN
	uiState:=NotReady;
END_IF

//	运行中
IF xRunning THEN
	uiState:=iRunning;
END_IF

//	报警中
IF xAlarm THEN
	uiState:=Alarm;
END_IF

//	准备好
IF xInitDone
	AND NOT xAlarm
	AND NOT xRunning
THEN
	uiState:=Ready;
END_IF

//工站完成
IF xInitDone AND xDone THEN 
	uiState:=Done;
END_IF
END_ACTION

ACTION ACT_Run:
//	运行条件
xRunAble:=xEStop
	AND xKey
	AND xSafety
	AND xInitDone
	AND NOT xAlarm
	AND NOT xAutoTip;

//	单动标志
ftCycleRunHMI(CLK:=xCycleRunHmi, Q=>);
rtJogRunHmi(CLK:=xJogRunHmi, Q=>);
IF xEStop
	AND xInitDone
THEN
	IF (ftCycleRunHMI.Q
			OR rtJogRunHmi.Q)
		AND xRunAble
		AND xManualMode
	THEN
		xSingleRunFlag:=TRUE;
	END_IF
ELSE
	xSingleRunFlag:=FALSE;
END_IF

//	连动中、寸动中
IF xRunAble
	AND xManualMode
	AND xSingleRunFlag
	AND NOT xPause
THEN
	IF ftCycleRunHMI.Q THEN
		xCycleRunning:=TRUE;
	END_IF
	xJogRunning:=rtJogRunHmi.CLK;
ELSE
	xCycleRunning:=FALSE;
	xJogRunning:=FALSE;
END_IF

//	单动中
xSingleRunning:=xCycleRunning
	OR xJogRunning;

//	运行中
xRunning:=xSingleRunning
	OR xMachineRunning
		AND xRunAble;

xDeviceRunning := xRunning OR xIniting;		
		
//工站自动流程超时

//ton_AutoTimeout(IN:= bRunning 
//					AND NOT bSingleRunFlag 
//					AND bCycleStart , PT:=T#35S , Q=> , ET=> );		//自动程序有BUG
END_ACTION

ACTION ACT_CycleTime:
//	初始化时同时初始化工站周期计时
IF xIniting THEN
	xCycleEnable:=FALSE;
END_IF

//工站完成触发信号
rStationStart(CLK:= xCycleEnable);
IF rStationStart.Q
THEN
	diCycleTime := 0;
END_IF
//	工站周期计时
IF xRunning AND xCycleEnable AND stSysPulse.xR100ms
THEN
	diCycleTime := diCycleTime + 1;//对应最小周期是0.1ms
END_IF
END_ACTION

ACTION ACT_General:
//	提示中
xAutoTip:=adwAutoTipOut[1]<>0 OR adwAutoTipOut[2]<>0 OR adwAutoTipOut[3]<>0 OR adwAutoTipOut[4]<>0;
xManualTip:=adwManualTipOut[1]<>0 OR adwManualTipOut[2]<>0 OR adwManualTipOut[3]<>0 OR adwManualTipOut[4]<>0;
xTip:=xAutoTip OR xManualTip;	
//	暂停
xPause:=xMachinePause
	OR xPauseHmi
	OR xStop;
//报警中
xAlarm:=adwAlarmOut[1]<>0 OR adwAlarmOut[2]<>0 OR adwAlarmOut[3]<>0 OR adwAlarmOut[4]<>0;

//	报警复位
IF xReset THEN
	FOR i:=1 TO 4 BY 1 DO 
		adwAutoTip[i] := adwAlarm[i] := adwManualTip[i] := 0;
	END_FOR
END_IF

//处理报警与提示信息,报警发生后，当当前报警消失且按下复位后，复位报警输出信号
IF NOT xDisabled THEN		 
	FOR i:=1 TO 4 BY 1 DO 
		FOR j:=0 TO 31 DO
			//报警
			IF GETBIT32(adwAlarm[i],j) THEN
				adwAlarmOut[i]:=TO_DWORD(CSETBIT32(adwAlarmOut[i],j,TRUE));
			ELSIF NOT GETBIT32(adwAlarm[i],j) AND xReset THEN 
				adwAlarmOut[i]:=TO_DWORD(CSETBIT32(adwAlarmOut[i],j,FALSE));			
			END_IF
		//自动提示
			IF GETBIT32(adwAutoTip[i],j) AND NOT xManualMode THEN
				adwAutoTipOut[i]:=TO_DWORD(CSETBIT32(adwAutoTipOut[i],j,TRUE));
			ELSIF NOT GETBIT32(adwAutoTip[i],j) AND xReset THEN 
				adwAutoTipOut[i]:=TO_DWORD(CSETBIT32(adwAutoTipOut[i],j,FALSE));			
			END_IF	
			//手动提示
			IF GETBIT32(adwManualTip[i],j) AND xManualMode THEN
				adwManualTipOut[i]:=TO_DWORD(CSETBIT32(adwManualTipOut[i],j,TRUE));
			ELSIF NOT GETBIT32(adwManualTip[i],j) AND xReset THEN 
				adwManualTipOut[i]:=TO_DWORD(CSETBIT32(adwManualTipOut[i],j,FALSE));			
			END_IF		
		END_FOR
	END_FOR
ELSE
	FOR i:=1 TO 4 BY 1 DO 
		FOR j:=0 TO 31 DO
				adwAlarmOut[i]:=TO_DWORD(CSETBIT32(adwAlarmOut[i],j,FALSE));
				adwAutoTipOut[i]:=TO_DWORD(CSETBIT32(adwAutoTipOut[i],j,FALSE));
				adwManualTipOut[i]:=TO_DWORD(CSETBIT32(adwManualTipOut[i],j,FALSE));	
		END_FOR
	END_FOR
END_IF

//将字转换为bool
FOR i:=1 TO 4 BY 1 DO
	FOR j:=0 TO 31 BY 1 DO
		xadwAutoTip[i,j]:=GETBIT32(adwAutoTipOut[i],j);
		xadwManualTip[i,j]:=GETBIT32(adwManualTipOut[i],j);
		xadwAlarm[i,j]:=GETBIT32(adwAlarmOut[i],j);
	END_FOR
END_FOR
END_ACTION

END_FUNCTION_BLOCK

// Device/Application/FB/50_CycleTime/FB_CycleTime
FUNCTION_BLOCK FB_CycleTime
VAR_INPUT	
	xCycleMark:BOOL;
	xCycleRun	:BOOL;
END_VAR
VAR_OUTPUT
	rCycleTime :REAL;
END_VAR
VAR
  StartTime,EndTime,ElapseTime :UDINT;	
END_VAR


//IF xCycleRun
//THEN
	IF xCycleMark
	THEN 
		GetSystemTime(udiTimeMs=> EndTime, uliTimeUs=> , uliTimeNs=> );	
		IF StartTime <> 0
		THEN 
			ElapseTime := EndTime-StartTime;
		END_IF
		GetSystemTime(udiTimeMs=> StartTime, uliTimeUs=> , uliTimeNs=> );
		xCycleMark:= FALSE;
	END_IF
//END_IF		
rCycleTime:= UDINT_TO_REAL(ElapseTime)/1000.0;

END_FUNCTION_BLOCK

// Device/Application/FB/11_AxisFB/FB_Axis
FUNCTION_BLOCK FB_Axis
VAR_INPUT
//	注意，倍福自带的伺服功能块需要隐藏，否则生成的TPY文件导入Proface后，FB_Axis不显示

	Basic_Axis					: ST_Axis_REF ;				//轴
	xEStop						: BOOL;					//急停
	xKey						: BOOL;					//钥匙开关
	xSafety						: BOOL;					//安全防护
	xManualMode					: BOOL;					//手动模式
	xAutoMode					: BOOL;					//自动模式
	xReset					: BOOL;					//报警复位,提示复位
	
	xHome					             	:BOOL;//原点
	xPositive					          :BOOL;//正极限
	xNegative					          :BOOL;//负极限
	xStop					         	: BOOL;					//轴停止
	xStopHmi					: BOOL;					//轴停止HMI
	xHalt						: BOOL;					//轴暂停
	xHaltHmi				    : BOOL;					//轴暂停HMI
	
	xEnablePositive 			: BOOL:=TRUE;			//允许正转
	xEnableNegative				: BOOL:=TRUE;			//允许反转
	xRunILC						: BOOL:=TRUE;			//运行条件
	
	xPowerHmi					: BOOL;					//使能手动HMI
	xPowerOff					: BOOL:=FALSE;;		    //使能关闭
	xBrakeHmi					: BOOL;					//刹车手动HMI
	xHomeHmi					: BOOL;					//原点搜索HMI
	xAlarmResetHmi				: BOOL;					//报警复位HMI
	
	xHomeILC                    : BOOL;                 //回原条件
	
	xJogILC                     : BOOL;                 //Jog条件
	xJogForwardHmi				: BOOL;					//Jog+HMI
	xJogBackwardsHmi			: BOOL;					//Jog-HMI
	
	xPowerInit					: BOOL;					//使能初始化执行
	xHomeAuto					: BOOL;					//原点搜索自动执行
	xCalibrationCam				: BOOL;					//原点校准
	xJogForwardAuto				: BOOL;					//Jog+自动执行
	xJogBackwardAuto			: BOOL;					//Jog-自动执行
	
	xMoveILC					: ARRAY[0..gc_uiAxisMoveNum] OF BOOL:=[TRUE];//绝对定位动作条件
	xMoveHmi					: ARRAY[0..gc_uiAxisMoveNum] OF BOOL;//绝对定位手动Hmi
	xMoveAuto					: ARRAY[0..gc_uiAxisMoveNum] OF BOOL;//绝对定位自动执行
	
	xRelativeILC                : BOOL;                 //Relative条件
	xRelativeHmi			    : BOOL;					//相对定位手动Hmi
	xRelativeAuto			    : BOOL;					//相对定位自动执行
	
	xVelocityILC                : BOOL;                 //Velocity条件
	xVelocityAuto			    : BOOL;					//连续运行启动
	xVelocityDirection          : BOOL;                 //连续运行方向  
	
	rMoveDiff			    	: ARRAY[0..gc_uiAxisMoveNum] OF  REAL:=[gc_uiAxisMoveNum(0.2)];	//轴定位误差
	rJogAcceleration            : REAL;                 //轴Jog加速度
	rJogDeceleration            : REAL;                 //轴Jog减速度
	rMoveAcceleration           : REAL;            //轴定位加速度                   	
	rMoveDeceleration           : REAL;           //轴定位减速度 
	rJogVelocity				:  REAL;	//轴Jog速度
	rManualVelocity				:  REAL;	//轴手动速度
	rAutoVelocity				:  REAL;	//轴自动速度
	rMovePosition				:  ARRAY[0..gc_uiAxisMoveNum] OF REAL;//绝对定位位置
	rMoveVelocity				:  ARRAY[0..gc_uiAxisMoveNum] OF REAL;//绝对定位速度
	tMoveInPos					:  ARRAY[0..gc_uiAxisMoveNum] OF TIME;//绝对定位到位延时
	rModuloHome					:  REAL;	//模长内定位初始角度
	tModuloInPos				:  TIME;	//模长内定位到位延时
	
	rRelativeDistance			: REAL;					//相对定位位置
	rRelativeVelocity			: REAL;					//相对定位速度
	
	rVelocityVel			    : REAL;					//连续运行速度
	rVelocityAcc			    : REAL;					//连续运行加速度
	rVelocityDec			    : REAL;					//连续运行减速度
	
	rStopDec                    : REAL:=0;              //停机减速度
	
	xModulo						: BOOL;					//模长内定位启动
	rModuloPosition				: REAL;					//模长内定位位置
	rModuloVelocity				: REAL;					//模长内定位速度
	iModuloDirection			: INT;					//模长定位方向
	tMoveTimeout				: TIME:=T#10S;			//定位超时
	byManualTip					: BYTE;					//手动提示字节，多个提示，用于外部触发
	xManualTip					: BOOL;					//手动提示，单个提示，用于外部触发

	
	xStopDone                   : BOOL;                 //停止完成信号
	
	xMoveDirection              : MC_DIRECTION ; //绝对定位方向
	iPosNumber					        : INT;					//位置保存编号
	lrHomeOffSet                : LREAL ; //原点偏置

END_VAR

VAR_OUTPUT
	xPowerOn					: BOOL;					//使能On
	xNotPowerOn					: BOOL;					//使能未On提示
    xBrakeUnlock			: BOOL;		//刹车打开状态
	xReady						: BOOL;					//准备好
	
	xPowerBusy					: BOOL;					//PowerBusy
	xPowerError					: BOOL;					//Power错误
	udiPowerErrorID				: UDINT;				//Power错误ID
	
	xJogDone					: BOOL;					//Jog定位完成
	xJogBusy					: BOOL;					//JogBusy
	xJogError					: BOOL;					//Jog错误
	udiJogErrorID					: UDINT;				//Jog错误ID
	
	xHomeDone					: BOOL;					//原点搜索完成
	xHomeBusy					: BOOL;					//原点搜索Busy
	xHomeError					: BOOL;					//原点搜索错误
	udiHomeErrorID				: UDINT;				//原点搜索错误ID
	
	xMoveInPos					: ARRAY[0..gc_uiAxisMoveNum] OF BOOL;//绝对定位到位
	xMoveDone					: ARRAY[0..gc_uiAxisMoveNum] OF BOOL;//绝对定位完成
	xMoveBusy					: ARRAY[0..gc_uiAxisMoveNum] OF BOOL;//绝对定位Busy
	xMoveError					: ARRAY[0..gc_uiAxisMoveNum] OF BOOL;//绝对定位错误
	udiMoveErrorID				: ARRAY[0..gc_uiAxisMoveNum] OF UDINT;//绝对定位错误ID
	
	xRelativeDone				: BOOL;					//相对定位完成
	xRelativeBusy				: BOOL;					//相对定位Busy
	xRelativeError				: BOOL;					//相对定位错误
	udiRelativeErrorID			: UDINT;				//相对定位错误ID
	
	xVelocityInVel				: BOOL;					//连续运行速度到达
	xVelocityBusy				: BOOL;					//连续运行Busy
	xVelocityError				: BOOL;					//连续运行错误
	udiVelocityErrorID			: UDINT;				//连续运行错误ID
	
	xModuloInPos				: BOOL;					//模长内定位到位
	xModuloDone					: BOOL;					//模长内定位完成
	xModuloBusy					: BOOL;					//模长内定位Busy
	xModuloError				: BOOL;					//模长内定位错误
	udiModuloErrorID			: UDINT;				//模长内定位错误ID
	
	xMoveTimeout				: BOOL;					//定位超时报警
	
	xError						: BOOL;					//错误
	xSwitch						: BOOL;					//软限位报错
	xbusy						: BOOL;
	udiErrorID					: UDINT;				//错误ID
	udiErrorCode				: UDINT;				//错误代码
	
	rSetTorque					: REAL;					//设定转矩
	rSetPos						: REAL;					//设定位置
	rModuloSetPos				: REAL;					//模长内定位设定位置
	rModuloSetTurns				: REAL;					//模长内定位设定匝数
	rTargetPos					: REAL;					//目标位置
	
	rActTorque					: REAL;					//当前转矩
	rActPos						: REAL;					//当前位置
	rActVelo					: REAL;					//当前速度
	rModuloActPos				: REAL;					//模长内定位当前位置
	rModuloActTurns				: REAL;					//模长内定位当前匝数
	rPosDiff					: REAL;					//跟随误差
	uiState						: UINT;					//状态
	xRelativeDone1				: BOOL;					//相对定位完成标志
END_VAR

VAR
	 
	ftPowerHmi					: F_TRIG;				//使能手动HMI下降沿
	{attribute 'hide'}
	 
	xPowerManual				: BOOL;					//使能手动执行
	{attribute 'hide'}
	 
	xPowerAuto					: BOOL;					//使能自动执行
	 {attribute 'hide'}
	xPowerEnable				: BOOL;					//使能Enable
	 {attribute 'hide'}
	rtPowerOn					: R_TRIG;				//使能上升沿
	 {attribute 'hide'}
	ftPowerOn					: F_TRIG;				//使能下降沿
	 {attribute 'hide'}
	tonNotPowerOn				: TON;					//伺服未On提示延时
	 {attribute 'hide'}
	ftBrakeHmi					: F_TRIG;				//刹车手动HMI下降沿
	 {attribute 'hide'}
	xRunable					: BOOL;					//可运行
	 {attribute 'hide'}
	ftHomeHmi					: F_TRIG;				//回原点HMI下降沿
	 {attribute 'hide'}
	xHomeManual					: BOOL;					//回原点手动执行
	 {attribute 'hide'}
	xHomeExecute				: BOOL;					//回原点触发
	 {attribute 'hide'}
	xJogForwardManual			: BOOL;					//Jog+手动执行
	 {attribute 'hide'}
	xJogBackwardManual			: BOOL;					//Jog-自动执行
	 {attribute 'hide'}
	xJogForward					: BOOL;					//Jog+
	 {attribute 'hide'}
	xJogBackward				: BOOL;					//Jog-
	 {attribute 'hide'}
	xMoveManual					: ARRAY[1..gc_uiAxisMoveNum] OF BOOL;//绝对定位手动执行
	 {attribute 'hide'}
	xMoveExecute				: ARRAY[1..gc_uiAxisMoveNum] OF BOOL;//绝对定位启动使能
	 {attribute 'hide'}
	xRelativeExecute			: BOOL;					//相对定位启动
	 {attribute 'hide'}
	xModuloExecute				: BOOL;					//模长内定位启动
	 {attribute 'hide'}
	xAnyMoveError				: BOOL;					//绝对定位故障
	 {attribute 'hide'}
	rVelocity					: REAL;					//定位速度
	 {attribute 'hide'}
	xVelocityExecute			: BOOL;					//相对定位启动
	 {attribute 'hide'}
	xVelocityAble			    : BOOL;					//相对定位启动
	 {attribute 'hide'}
	tonMoveInPos				: ARRAY[1..gc_uiAxisMoveNum] OF TON;//绝对定位到位计时
	 {attribute 'hide'}
	tonMoveTimeout				: ARRAY[1..gc_uiAxisMoveNum] OF TON;//绝对定位超时
	 {attribute 'hide'}
	tonModuloInPos				: TON;					//模长内定位到位计时
	 {attribute 'hide'}
	tonRelativeTimeout			: TON;					//相对定位超时
	 {attribute 'hide'}
	tonModuloTimeout			: TON;					//模长内定位超时
	 {attribute 'hide'}
	nIndexMove					: INT;					//绝对定位索引
	 {attribute 'hide'}
	xHaltExecute				: BOOL;					//轴暂停
	 {attribute 'hide'}
	xStopExecute				: BOOL;					//轴停止
	 {attribute 'hide'}
	bResetMove					: ARRAY[0..gc_uiAxisMoveNum] OF BOOL;//绝对定位启动复位
	{attribute 'hide'}
	rtbRelativeDone				: R_TRIG;				//相对定位完成标志 robert
	{attribute 'hide'}
  iIndex : INT;
	{attribute 'hide'}
END_VAR
VAR
	fbReadStatus				: MC_ReadStatus;		//读取状态功能块
{attribute 'hide'}
	fbPower						: MC_Power;				//使能功能块
{attribute 'hide'}
	fbJog						: MC_Jog;				//Jog功能块
{attribute 'hide'}
	fbHome						: MC_Home;				//原点搜索功能块
{attribute 'hide'}
	fbMove						: ARRAY[0..gc_uiAxisMoveNum] OF MC_MoveAbsolute;//绝对定位功能块
{attribute 'hide'}
	fbRelative					: MC_MoveRelative;		//相对定位功能块
{attribute 'hide'}
	fbReset						: HMC_ResetServo;				//错误复位功能块
{attribute 'hide'}
	fbHalt						: MC_Halt;				//轴暂停功能块
{attribute 'hide'}
	fbStop						: MC_Stop;				//轴停止功能块
{attribute 'hide'}
	fbVelocity					: MC_MoveVelocity;	    //轴速度运行功能块
{attribute 'hide'}
	fbResetServo			    : HMC_ResetServo;    //轴速度运行功能块
	{attribute 'hide'}
END_VAR


ACT_ReadStatus();
ACT_Power();
ACT_Jog();
ACT_Home();
ACT_Move();
ACT_Relative();
ACT_InPos();
ACT_Timeout();
ACT_Tip();
ACT_Reset();
ACT_Halt();
ACT_Stop();
ACT_Velocity();
ACT_ReinitDrive();

//自动复位，无需程序里做初始化
xStop:=FALSE;
xHalt:=FALSE;
xReset:=FALSE;
xPowerInit:=FALSE;
//xPowerOff:=FALSE;
xModulo:=FALSE;
xMoveAuto:=bResetMove;
//xHomeAuto:=FALSE;
(*IF NOT xAutoMode
THEN

	xJogForwardAuto:=FALSE;
	xJogBackwardAuto:=FALSE;
END_IF
*)
FOR iIndex:=1 TO gc_uiAxisMoveNum DO
	xMoveHmi[iIndex]:=FALSE;
	xMoveAuto[iIndex]:=FALSE;
END_FOR
xRelativeAuto:=FALSE;
//bVelocityAuto:=FALSE;//在自动流程里RST
///////////////////////////////////////////////

ACTION ACT_Tip:
IF xReset THEN
	xManualTip:=
	xNotPowerOn:=FALSE;
	xManualTip:=0;
END_IF

tonNotPowerOn(
	IN:=NOT xPowerOn
		AND xPowerAuto,
	PT:=T#3S,
	Q=> , ET=>
);
IF tonNotPowerOn.Q
	AND xAutoMode
	AND NOT Basic_Axis.Axis^.bError
THEN
	xNotPowerOn:=TRUE;
END_IF
END_ACTION

ACTION ACT_Move:
FOR nIndexMove:=1 TO gc_uiAxisMoveNum DO
	IF xAutoMode THEN
		IF rMoveVelocity[nIndexMove]>0 THEN
			rVelocity:=rMoveVelocity[nIndexMove];
		ELSE
			rVelocity:=rAutoVelocity;
		END_IF
	ELSE
		rVelocity:=rManualVelocity;
	END_IF
	xMoveManual[nIndexMove]:=xMoveHmi[nIndexMove]
		AND xManualMode;
	xMoveExecute[nIndexMove]:=xRunable
		AND xMoveILC[nIndexMove]
		AND (xMoveManual[nIndexMove]
			OR xMoveAuto[nIndexMove]);
	fbMove[nIndexMove](
		Axis:=Basic_Axis.Axis^,
		Execute:=xMoveExecute[nIndexMove],
		Position:=REAL_TO_LREAL(rMovePosition[nIndexMove]),
		Velocity:=REAL_TO_LREAL(rVelocity),
		Acceleration:=rMoveAcceleration,
		Deceleration:=rMoveDeceleration,
		Direction:=xMoveDirection,
		Jerk:=0,
		Done=>xMoveDone[nIndexMove],
		Busy=>xMoveBusy[nIndexMove],
		CommandAborted=>,
		Error=>,
		ErrorID=>
	);
END_FOR
//判断旋转方向
END_ACTION

ACTION ACT_Reset:

fbReset(
	Axis:= Basic_Axis.Axis^, 
	Slave:= Basic_Axis.Server^ , 
	xExecute:= (xReset OR xAlarmResetHmi) AND xError AND Basic_Axis.Axis^.wCommunicationState=100, 
	xDone=> , 
	xBusy=> , 
	xError=> , 
	eErrorID=> );
END_ACTION

ACTION ACT_Halt:
 
xHaltExecute:=xRunable
		AND ((xHaltHmi AND xManualMode) OR (xHalt AND xAutoMode));
fbHalt(
	Axis:=Basic_Axis.Axis^,
	Execute:=xHaltExecute,
	Deceleration:=100000,
	Jerk:=,
	Done=>,
	Busy=>,
	CommandAborted=>,
	Error=>,
	ErrorID=>
);
END_ACTION

ACTION ACT_ReinitDrive:
 


fbResetServo(
	Axis:=Basic_Axis.Axis^ , 
	Slave:=Basic_Axis.Server^ , 
	xExecute:=xReset AND Basic_Axis.Axis^.wCommunicationState<>100, 
	xDone=> , 
	xBusy=> , 
	xError=> , 
	eErrorID=> );
END_ACTION

ACTION ACT_Home:
 
ftHomeHmi(CLK:=xHomeHmi, Q=>);
xHomeManual:=ftHomeHmi.Q
	AND xManualMode;
xHomeExecute:=xRunable
	AND xHomeILC
    AND(xHomeManual
		OR xHomeAuto);
fbHome(
	Axis:=Basic_Axis.Axis^,
	Execute:=xHomeExecute ,
	Position:=lrHomeOffSet,
	Done=>xHomeDone,
	Busy=>,
	CommandAborted=>,
	Error=>,
	ErrorID=>
);
END_ACTION

ACTION ACT_Stop:
 
IF rStopDec<=0 THEN
  fbStop.Deceleration:=100000;
ELSE
  fbStop.Deceleration:=REAL_TO_LREAL(rStopDec);	
END_IF
xStopExecute:=xRunable
		AND ((xStopHmi AND xManualMode) OR xStop);// AND xAutoMode));
fbStop(
	Axis:=Basic_Axis.Axis^,
	Execute:=xStopExecute,
	Deceleration:= ,
	Jerk:=,
	Done=>xStopDone,
	Busy=>,
	Error=>,
	ErrorID=>
);
END_ACTION

ACTION ACT_Jog:
xJogForwardManual:=xJogForwardHmi
	AND xManualMode;
xJogBackwardManual:=xJogBackwardsHmi
	AND xManualMode;
xJogForward:=xRunable
    AND xJogILC
	AND NOT xJogBackward
	AND (xJogForwardManual
		OR xJogForwardAuto);
xJogBackward:=xRunable
    AND xJogILC
	AND NOT xJogForward
	AND (xJogBackwardManual
		OR xJogBackwardAuto);

fbJog(
	Axis:=Basic_Axis.Axis^,
	JogForward:=xJogForward,
	JogBackward:=xJogBackward,
	Velocity:=REAL_TO_LREAL(rJogVelocity),
	Acceleration:=rJogAcceleration,
	Deceleration:=rJogDeceleration,
	Jerk:=0,
	Busy=>xJogBusy,
	CommandAborted=>,
	Error=>,
	ErrorID=>
);
END_ACTION

ACTION ACT_Timeout:
IF xReset THEN
	xMoveTimeout:=FALSE;
END_IF

tonRelativeTimeout(
	IN:=xRelativeAuto,
	PT:=tMoveTimeout,
	Q=>, ET=>);
IF tonRelativeTimeout.Q THEN
	xMoveTimeout:=TRUE;
END_IF

tonModuloTimeout(
	IN:=xModulo
		AND NOT xModuloInPos,
	PT:=tMoveTimeout,
	Q=>, ET=>);
IF tonModuloTimeout.Q THEN
	xMoveTimeout:=TRUE;
END_IF

IF NOT xMoveTimeout THEN
	FOR nIndexMove:=1 TO gc_uiAxisMoveNum DO
		tonMoveTimeout[nIndexMove](
			IN:=xMoveAuto[nIndexMove]
				AND NOT xMoveInPos[nIndexMove],
			PT:=tMoveTimeout,
			Q=>, ET=>);
		IF tonMoveTimeout[nIndexMove].Q THEN
			xMoveTimeout:=TRUE;
			EXIT;
		END_IF
	END_FOR
END_IF
END_ACTION

ACTION ACT_Power:
ftPowerHmi(CLK:=xPowerHmi, Q=>);
IF xEStop THEN
	IF ftPowerHmi.Q
		AND xKey
		AND xSafety
		AND xManualMode
	THEN
		xPowerManual:=NOT xPowerManual;
	END_IF
	IF xPowerInit  THEN 
		xPowerManual:=FALSE;
		xPowerAuto:=TRUE;
	END_IF
ELSE
	xPowerManual:=FALSE;
	xPowerAuto:=FALSE;
END_IF
xPowerEnable:=NOT Basic_Axis.Axis^.bError
	AND (xPowerManual
		XOR xPowerAuto);
fbPower(
	Axis:=Basic_Axis.Axis^,
	Enable:=TRUE,
	bRegulatorOn:=xPowerEnable AND NOT xPowerOff ,
	bDriveStart:=xPowerEnable AND NOT xPowerOff,
	Status=>xPowerOn,
	Busy=>,
	Error=>,
	ErrorID=>
);
xReady:=xPowerOn
	AND NOT Basic_Axis.Axis^.bError
	AND Basic_Axis.Axis^.bCommunication;
xRunable:=xEStop
	AND xKey
	AND xSafety
	AND xReady
	AND xRunILC;
END_ACTION

ACTION ACT_Relative:
IF xAutoMode THEN
	IF rRelativeVelocity>0 THEN
		rVelocity:=rRelativeVelocity;
	ELSE
		rVelocity:=rAutoVelocity;
	END_IF
ELSE
	rVelocity:=rManualVelocity;
END_IF
xRelativeExecute:=xRunable
		AND ((xRelativeHmi AND xManualMode) OR xRelativeAuto ) AND xRelativeILC;

fbRelative(
	Axis:=Basic_Axis.Axis^,  
	Execute:= xRelativeExecute, 
	Distance:= REAL_TO_LREAL(rRelativeDistance), 
	Velocity:= REAL_TO_LREAL(rVelocity), 
	Acceleration:= rMoveAcceleration, 
	Deceleration:= rMoveDeceleration, 
	Jerk:= , 
	Done=> xRelativeDone, 
	Busy=> xRelativeBusy, 
	CommandAborted=> , 
	Error=> xRelativeError, 
	ErrorID=> udiRelativeErrorID);	

IF xRelativeDone=TRUE THEN
	xRelativeDone1:=TRUE;
ELSIF xRelativeBusy=TRUE THEN
	xRelativeDone1:=FALSE;	
END_IF//
END_ACTION

ACTION ACT_InPos:
//	绝对定位到位
FOR nIndexMove:=1 TO gc_uiAxisMoveNum DO
	tonMoveInPos[nIndexMove](
		IN:=xReady
			AND Basic_Axis.Axis^.nAxisState=3
			AND Basic_Axis.Axis^.fActPosition > REAL_TO_LREAL(rMovePosition[nIndexMove]) - rMoveDiff[nIndexMove]
			AND Basic_Axis.Axis^.fActPosition < REAL_TO_LREAL(rMovePosition[nIndexMove]) + rMoveDiff[nIndexMove] ,
		PT:=tMoveInPos[nIndexMove],
		Q=>xMoveInPos[nIndexMove],
		ET=>);
END_FOR
END_ACTION

ACTION ACT_Velocity:
IF xAutoMode THEN
	IF rVelocityVel>0 THEN
		fbVelocity.Velocity:=rVelocityVel;
	ELSE
		fbVelocity.Velocity:=rAutoVelocity;
	END_IF
ELSE
	fbVelocity.Velocity:=rManualVelocity;
END_IF
xVelocityExecute:=xRunable AND xVelocityAuto AND xVelocityILC;


fbVelocity(
	Axis:=Basic_Axis.Axis^ , 
	Execute:=xVelocityExecute AND xVelocityAble , 
	Velocity:= , 
	Acceleration:=rVelocityAcc , 
	Deceleration:=rVelocityDec , 
	Jerk:= , 
	Direction:= , 
	InVelocity=>xVelocityInVel , 
	Busy=>xVelocityBusy , 
	CommandAborted=> , 
	Error=>xVelocityError , 
	ErrorID=>udiVelocityErrorID );
xVelocityAble:= NOT xVelocityAble;
END_ACTION

ACTION ACT_ReadStatus:
fbReadStatus(
	Axis:=Basic_Axis.Axis^,
	Enable:=TRUE,
	Valid=>,
	Busy=>,
	Error=>,
	ErrorID=>,
	ErrorStop=>,
	Disabled=>,
	Stopping=>,
	StandStill=>,
	DiscreteMotion=>,
	ContinuousMotion=>,
	SynchronizedMotion=>,
	Homing=>,
	ConstantVelocity=>,
	Accelerating=>,
	Decelerating=>,
);

xAnyMoveError:=FALSE;
FOR nIndexMove:=1 TO gc_uiAxisMoveNum DO
	xAnyMoveError S=(xMoveError[nIndexMove]);
END_FOR
xError					:=Basic_Axis.Axis^.nAxisState=1 OR Basic_Axis.Axis^.bError OR xSwitch OR (
                          fbHalt.Error OR fbhome.Error OR fbjog.Error OR 
                          fbpower.Error OR fbrelative.Error OR fbReset.xError  OR 
                          fbstop.Error OR fbvelocity.Error OR xAnyMoveError) ;
xSwitch        			:=Basic_Axis.Axis^.usiSWEndSwitchState =2;//软限位
udiErrorID				:=Basic_Axis.Axis^.dwErrorID;
xbusy					:=Basic_Axis.Axis^.nAxisState>3;
//nErrorCode				:=Axis.NcToPlc.ErrorCode;需要读200B-23h
IF xSwitch
THEN 
  udiErrorID := 1;
END_IF
rSetTorque				:=LREAL_TO_REAL(Basic_Axis.Axis^.fSetTorque);
rSetPos					:=LREAL_TO_REAL(Basic_Axis.Axis^.fSetPosition);
rTargetPos				:=LREAL_TO_REAL(Basic_Axis.Axis^.fAimPosition);

rActTorque				:=LREAL_TO_REAL(Basic_Axis.Axis^.fActTorque);
rActPos					:=LREAL_TO_REAL(Basic_Axis.Axis^.fActPosition);
rActVelo				:=LREAL_TO_REAL(Basic_Axis.Axis^.fActVelocity);
rPosDiff				:=LREAL_TO_REAL(Basic_Axis.Axis^.fFollowingError);

xHome    :=Basic_Axis.Axis^.in.dwDigitalInputs.2;
xPositive:=Basic_Axis.Axis^.in.dwDigitalInputs.1;
xNegative:=Basic_Axis.Axis^.in.dwDigitalInputs.0;
END_ACTION

END_FUNCTION_BLOCK

// Device/Application/FB/10_CylinderFB/FB_Cylinder
FUNCTION_BLOCK FB_Cylinder
VAR_INPUT
	xEStop						: BOOL;					//急停
	xSafety						: BOOL;					//安全防护
	xManualMode					: BOOL;					//手动模式
	xAutoMode					: BOOL;					//自动模式
	xAirOn						: BOOL;					//气压正常
	tAlarm						: TIME:=T#5S;			//报警延时
	xReset					: BOOL;					//报警复位,提示复位
	xAlarmDisable               : BOOL;                 //报警屏蔽
	
	xHmi						: BOOL;					//手动HMI按钮
	xManual						: BOOL;					//手动执行
	xAuto						: BOOL;					//自动执行
	xInit						: BOOL;					//初始化执行
	xRelease					: BOOL;					//输出释放，气缸泄气
	xOnILC						: BOOL;			        //动作条件
	xOffILC						: BOOL;			        //复位条件
	xHP_Sensor					: BOOL;					//原点感应器
	xWP_Sensor					: BOOL;					//动点感应器
	tHP_Delay					: TIME;	//原点延时
	tWP_Delay					: TIME;	//动点延时
	byManualTip					: BYTE;					//手动提示字节，多个提示，用于外部触发
	xManualTip					: BOOL;					//手动提示，单个提示，用于外部触发
END_VAR

VAR_OUTPUT
	xHP_Valve					: BOOL;					//原点阀
	xWP_Valve					: BOOL;					//动点阀
	xHP_Delay					: BOOL;					//原点状态
	xWP_Delay					: BOOL;					//动点状态
	xHP_Off						: BOOL;					//原点无信号
	xWP_Off						: BOOL;					//动点无信号
	xHP_On						: BOOL;					//原点应为Off
	xWP_On						: BOOL;					//动点应为Off
	xAutoTip					: BOOL;					//自动提示，用于外部触发
	xAlarming					: BOOL;					//报警中
	xBusy						: BOOL;					//运动中
END_VAR

VAR
	 
	ftHmi						: F_TRIG;				//手动HMI下降沿
	{attribute 'hide'}
	 
	rtManual					: R_TRIG;				//手动执行上升沿
	{attribute 'hide'}
//	 
	xEnable						: BOOL;					//使能
	{attribute 'hide'}
	 
	tonHP_Delay					: TON;					//原点延时计时
	{attribute 'hide'}
	 
	tonWP_Delay					: TON;					//动点延时计时
	{attribute 'hide'}
	 
	tAlarmTime					: TIME;					//报警延时
	{attribute 'hide'}
	 
	tonHP						: TON;					//原点输出计时
	{attribute 'hide'}
	 
	tonWP						: TON;					//动点输出计时
	{attribute 'hide'}
END_VAR

ACT_Manual();
ACT_Output();
ACT_Delay();
ACT_Alarm();
ACT_Tip();

//	自动复位
xInit:=FALSE;
xHmi:=FALSE;

ACTION ACT_Delay:
//	原点延时
tonHP_Delay(
	IN:=xHP_Valve
		AND NOT xWP_Valve
		AND xHP_Sensor
		AND NOT xWP_Sensor,
	PT:=tHP_Delay,
	Q=>xHP_Delay,
	ET=>);

//	动点延时
tonWP_Delay(
	IN:=NOT xHP_Valve
		AND xWP_Valve
		AND NOT xHP_Sensor
		AND xWP_Sensor,
	PT:=tWP_Delay,
	Q=>xWP_Delay,
	ET=>);
END_ACTION

ACTION ACT_Output:
//	使能
rtManual(CLK:=xManual, Q=> );
IF xEStop THEN
	IF rtManual.Q		OR xInit
	THEN
		xEnable:=TRUE;
	END_IF
ELSE
	;//xEnable:=FALSE;
END_IF

//	原点阀输出
xHP_Valve:=xEnable	AND NOT xRelease	AND (xManual = xAuto)AND xOffILC;

//	动点阀输出
xWP_Valve:=xEnable	AND NOT xRelease	AND (xManual XOR xAuto)AND xOnILC;
END_ACTION

ACTION ACT_Tip:
IF xReset THEN
	xManualTip:=FALSE;
	byManualTip:=0;
END_IF

xAutoTip:=xAutoMode AND xManual;
END_ACTION

ACTION ACT_Manual:
//	手动操作
ftHmi(CLK:=xHmi, Q=>);
IF ftHmi.Q	AND xEStop	AND xSafety	AND xManualMode	AND xAirOn	AND ((xManual = xAuto	AND xOnILC)		OR ((xManual XOR xAuto)	AND xOffILC		)	)
THEN
	xManual:=NOT xManual;
END_IF

//	初始化时复位手动执行//复位自动执行
IF xInit THEN
	xManual:=FALSE;
	xAuto  :=FALSE;
END_IF
END_ACTION

ACTION ACT_Alarm:
//	延时设置，防止报警延时小于到位延时误报警
IF tAlarm > MAX(tHP_Delay, tWP_Delay) THEN
	tAlarmTime:=tAlarm;
ELSE
	tAlarmTime:=tAlarm + MAX(tHP_Delay, tWP_Delay);
END_IF

//	报警延时
tonHP(IN:=xAirOn AND xHP_Valve, PT:=tAlarmTime, Q=>, ET=>);
tonWP(IN:=xAirOn AND xWP_Valve, PT:=tAlarmTime, Q=>, ET=>);

//	先报警复位
IF xReset THEN
	 xHP_Off:=FALSE;
	 xWP_Off:=FALSE;
	 xHP_On:=FALSE;
	 xWP_On:=FALSE;
END_IF

//	报警输出，Off报警用延时，On报警用感应器，防止感应器抖动时无到位无报警
IF tonHP.Q AND NOT xAlarmDisable THEN
	IF NOT xHP_Delay THEN
		xHP_Off:=TRUE;
	END_IF
	IF xWP_Sensor THEN
		xWP_On:=TRUE;
	END_IF
END_IF

IF tonWP.Q AND NOT xAlarmDisable THEN
	IF NOT xWP_Delay THEN
		xWP_Off:=TRUE;
	END_IF
	IF xHP_Sensor THEN
		xHP_On:=TRUE;
	END_IF
END_IF

xAlarming:=(xHP_Off OR xWP_Off OR xHP_On OR xWP_On) AND NOT xAlarmDisable;

xBusy:=NOT xAlarming
	AND (xHP_Valve AND NOT xHP_Delay
		OR xWP_Valve AND NOT xWP_Delay);
END_ACTION

END_FUNCTION_BLOCK

// Device/Application/FB/50_CycleTime/FB_CycleTime_1
FUNCTION_BLOCK FB_CycleTime_1
VAR_INPUT	
	xCycleMark:BOOL;
	xCycleRun	:BOOL;
END_VAR
VAR_OUTPUT
	rCycleTime :REAL;
END_VAR
VAR
  StartTime,EndTime,ElapseTime :UDINT;	
  Rt_Ctmark             :R_TRIG;
  Ft_Ctmark             :F_TRIG;
END_VAR

Rt_Ctmark(CLK:=xCycleMark, Q=> ); 
Ft_Ctmark(CLK:=xCycleMark, Q=> ); 
//IF xCycleRun
//THEN
	IF Ft_Ctmark.Q	THEN 
		GetSystemTime(udiTimeMs=> EndTime, uliTimeUs=> , uliTimeNs=> );	
  END_IF
	IF Rt_Ctmark.Q	THEN 
		GetSystemTime(udiTimeMs=> StartTime, uliTimeUs=> , uliTimeNs=> );
	END_IF
	IF Ft_Ctmark.Q THEN 
	ElapseTime := EndTime-StartTime;
	END_IF
//END_IF		
rCycleTime:= UDINT_TO_REAL(ElapseTime)/1000.0;

END_FUNCTION_BLOCK

// Device/Application/FB/50_CycleTime/FB_CycleTime_2
FUNCTION_BLOCK FB_CycleTime_2
VAR_INPUT	
	xCycleStartMark:BOOL;
	xCycleEndMark:BOOL;
	xCycleRun	:BOOL;
END_VAR
VAR_OUTPUT
	rCycleTime :REAL;
END_VAR
VAR
  StartTime,EndTime,ElapseTime :UDINT;	
  Rt_Ctstartmark             :R_TRIG;
  Rt_Ctendmark               :R_TRIG;
END_VAR

Rt_Ctstartmark(CLK:=xCycleStartMark, Q=> ); 
Rt_Ctendmark(CLK:=xCycleEndMark, Q=> ); 
//IF xCycleRun
//THEN
	IF Rt_Ctendmark.Q	THEN 
		GetSystemTime(udiTimeMs=> EndTime, uliTimeUs=> , uliTimeNs=> );	
  END_IF
	IF Rt_Ctstartmark.Q	THEN 
		GetSystemTime(udiTimeMs=> StartTime, uliTimeUs=> , uliTimeNs=> );
	END_IF
	IF Rt_Ctendmark.Q THEN 
	ElapseTime := EndTime-StartTime;
	END_IF
//END_IF		
rCycleTime:= UDINT_TO_REAL(ElapseTime)/1000.0;

END_FUNCTION_BLOCK

// Device/Application/POUS/02_STATION/S01_transplant
PROGRAM S01_transplant
VAR_INPUT
//工站
	station					    : REFERENCE TO FB_Station:=fbStation[1];//工站状态
	cycleTime						: REFERENCE TO FB_CycleTime:= fbStCycleTime[1];	//工站CT

//气缸
	Cy_rotate				    : REFERENCE TO FB_Cylinder:=fbCylinder[1];//旋转气缸
	Cy_takeClamp1				    : REFERENCE TO FB_Cylinder:=fbCylinder[2];//夹爪1 -B-H
//	Cy_takeClamp2				    : REFERENCE TO FB_Cylinder:=fbCylinder[3];//夹爪2-A-H
	Cy_takeClamp3				    : REFERENCE TO FB_Cylinder:=fbCylinder[4];//夹爪3-A-W
//	Cy_takeClamp4				    : REFERENCE TO FB_Cylinder:=fbCylinder[5];//夹爪4-B-W
  Cy_lifter			            : REFERENCE TO FB_Cylinder:=fbCylinder[6];//升降气缸
	//传感器
	Sensor_CV_on                   : ARRAY[0..2] OF BOOL; //传送带到位信号
	Sensor_Cycleline_on            : ARRAY[0..2] OF BOOL; //环形线放置到位
  

END_VAR
//内部变量
VAR
			arTon                 :ARRAY[0..10] OF ton ; 
	   	arTon_alarm           :ARRAY[0..10] OF ton ; 
			Cy_rotate_on          :BOOL ;//旋转气缸到位
		  rt_Ctmark             :R_TRIG;
  	  rt_Clamp1HP           :R_TRIG;
	    rt_Clamp2HP           :R_TRIG;
		  ft_cv                 :F_TRIG;
			CT_DisAction          : ARRAY[0..10] OF FB_CycleTime;
			CT_DisAction_1        : ARRAY[0..10] OF FB_CycleTime_1;			
	  	CT_DisAction_2        : ARRAY[0..10] OF FB_CycleTime_2;	
			Rt_Alarm              : ARRAY[0..31] OF R_TRIG;
			iLiferDown_can        : INT;
END_VAR

Alarm();
Delay();
FlowAuto();
FlowInit();
General();
ILC();
TipAuto();
TipManual();

ACTION TipManual:
//--------------------------------------------ManualTip------------------------------------------------------
station.adwManualTip[1].00			:=FALSE;//提示1
//-------------------------------------------气缸提示---------------------------------------------------------




/////////////////////////////////////////////////////////////////////////////////////////////////////////////////
END_ACTION

ACTION General:
//旋转气缸到位判断
IF Cy_rotate.xHP_Sensor OR Cy_rotate.xWP_Sensor THEN
	Cy_rotate_on:=TRUE;
END_IF

//----------------------------------CT-----------------------------------
rt_Ctmark(CLK:=Cy_rotate_on , Q=>cycleTime.xCycleMark );


CT_DisAction_2[1](xCycleStartMark:=Cy_lifter.xHP_Valve ,xCycleEndMark:= Cy_lifter.xHP_Delay,xCycleRun:=TRUE, RCycleTime=>ct_show.S01_CY_Lifter_HP);
CT_DisAction_2[2](xCycleStartMark:=Cy_lifter.xWP_Valve ,xCycleEndMark:= Cy_lifter.xWP_Delay,xCycleRun:=TRUE, RCycleTime=>ct_show.S01_CY_Lifter_WP);
CT_DisAction_2[3](xCycleStartMark:=Cy_rotate.xHP_Valve ,xCycleEndMark:= Cy_rotate.xHP_Delay,xCycleRun:=TRUE, RCycleTime=>ct_show.S01_CY_Rotate_HP);
CT_DisAction_2[4](xCycleStartMark:=Cy_rotate.xWP_Valve ,xCycleEndMark:= Cy_rotate.xWP_Delay,xCycleRun:=TRUE, RCycleTime=>ct_show.S01_CY_Rotate_WP);
CT_DisAction_2[5](xCycleStartMark:=Cy_takeClamp1.xHP_Valve ,xCycleEndMark:= Cy_takeClamp1.xHP_Delay,xCycleRun:=TRUE, RCycleTime=>ct_show.S01_Cy_takeClamp12_HP);
CT_DisAction_2[6](xCycleStartMark:=Cy_takeClamp1.xWP_Valve ,xCycleEndMark:= Cy_takeClamp1.xWP_Delay,xCycleRun:=TRUE, RCycleTime=>ct_show.S01_Cy_takeClamp12_WP);
CT_DisAction_2[7](xCycleStartMark:=Cy_takeClamp3.xHP_Valve ,xCycleEndMark:= Cy_takeClamp3.xHP_Delay,xCycleRun:=TRUE, RCycleTime=>ct_show.S01_Cy_takeClamp34_HP);
CT_DisAction_2[8](xCycleStartMark:=Cy_takeClamp3.xWP_Valve ,xCycleEndMark:= Cy_takeClamp3.xWP_Delay,xCycleRun:=TRUE, RCycleTime=>ct_show.S01_Cy_takeClamp34_WP);
CT_DisAction_2[9](xCycleStartMark:=station.iStepAuto= 5 AND NOT station.xDone ,xCycleEndMark:= station.xDone, RCycleTime=>ct_show.S01_Total);
//---------------------------------CV运行---------------------------------
 IF Machine_IO.xAutoMode THEN //自动模式下
	 IF station.xRunning THEN
		  Motion_cv_run[1]:=TRUE;//传送带运行置位
      Motion_cv_run[2]:=TRUE;   
   END_IF
END_IF
ft_cv(CLK:=station.xRunning AND  Machine_IO.xAutoMode , Q=> );
IF ft_cv.Q THEN
	 Motion_cv_run[1]:=FALSE;//传送带运行复位
   Motion_cv_run[2]:=FALSE;  
 END_IF
 
 //--------------------------------数据处理------------------------------
  rt_Clamp1HP(CLK:=Cy_takeClamp1.xHP_Delay, Q=> );
  rt_Clamp2HP(CLK:=Cy_takeClamp3.xHP_Delay , Q=> );
 //IF (rt_Clamp1HP.Q AND  Cy_rotate.xWP_Sensor) OR (rt_Clamp2HP.Q AND Cy_rotate.xHP_Sensor) THEN 	     
 IF station.xRunning AND NOT S05_CircleLine.Axis_Cycleline.xbusy THEN
   IF	 Sensor_Cycleline_on[1] OR (fbmachine[1].xTryRun) THEN
		 CardState[1].A:=TRUE;
		 CardState[1].Card_OK:=TRUE;	
   END_IF
   IF	 Sensor_Cycleline_on[2] OR (fbmachine[1].xTryRun) THEN
	 	 CardState[1].B:=TRUE;
		 CardState[1].Card_OK:=TRUE;	
	 END_IF
END_IF
 //--------------------------------下降与载具环形线互锁------------------------------
IF iLiferDown_can=1 AND Cy_rotate_on AND NOT S05_CircleLine.Axis_Cycleline.xbusy  THEN 
	iLiferDown_can:=2;
END_IF
END_ACTION

ACTION Delay:

//----------------------------------------------动作延时-----------------------------------------------

arTon[1](IN:=(Sensor_CV_on[1] AND NOT Sensor_CV_on[2]) OR (NOT Sensor_CV_on[1] AND  Sensor_CV_on[2])  , PT:=T#10S , Q=> , ET=> );//单个料延时取料
arTon[2](IN:=   , PT:=T#60S , Q=> , ET=> );//
arTon[3](IN:=   , PT:=T#60S , Q=> , ET=> );//


//----------------------------------------------报警延时-----------------------------------------------
arTon_alarm[1](IN:= , PT:=T#7S , Q=> , ET=> );//
arTon_alarm[2](IN:= , PT:=T#7S , Q=> , ET=> );//
arTon_alarm[3](IN:= , PT:=T#7S , Q=> , ET=> );//
arTon_alarm[4](IN:= , PT:=T#7S , Q=> , ET=> );//
arTon_alarm[5](IN:=   , PT:=T#60S , Q=> , ET=> );//
arTon_alarm[6](IN:=   , PT:=T#60S , Q=> , ET=> );//

arTon_alarm[7](IN:=   , PT:=T#10S , Q=> , ET=> );//
arTon_alarm[8](IN:=   , PT:=T#60S , Q=> , ET=> );//
arTon_alarm[9](IN:=   , PT:=T#60S , Q=> , ET=> );//
END_ACTION

ACTION Alarm:
station.adwAlarm[1].00:=station.xInitTimeout;	             //工站初始化超时报警

station.adwAlarm[1].01:=	Cy_rotate.xHP_Off ;        
station.adwAlarm[1].02:=	Cy_rotate.xWP_Off ;        
station.adwAlarm[1].03:=	Cy_takeClamp1.xHP_Off ;        //
station.adwAlarm[1].04:=	Cy_takeClamp1.xWP_Off ;        //
//station.adwAlarm[1].05:=	Cy_takeClamp2.xHP_Off ;        //
//station.adwAlarm[1].06:=	Cy_takeClamp2.xWP_Off ;        //
station.adwAlarm[1].07:=	Cy_takeClamp3.xHP_Off ;        //
station.adwAlarm[1].08:=	Cy_takeClamp3.xWP_Off;         //
//station.adwAlarm[1].09:=	Cy_takeClamp4.xHP_Off;         //
//station.adwAlarm[1].10:=	Cy_takeClamp4.xWP_Off ;        //
station.adwAlarm[1].11:=	Cy_lifter.xHP_Off ;        //
station.adwAlarm[1].12:=	Cy_lifter.xWP_Off ;        //
END_ACTION

ACTION TipAuto:

//------------------------------------------------AutoTip General---------------------------------


//------------------------------------------------AutoTip Cylinder--------------------------------

station.adwAutoTip[1].00:=FALSE;	//
station.adwAutoTip[1].01:=FALSE;	//
station.adwAutoTip[1].02:=Cy_rotate.xAutoTip;	       //Cy_rotate 气缸自动中有手动
station.adwAutoTip[1].03:=Cy_takeClamp1.xAutoTip;	   //Cy_takeClamp1 气缸自动中有手动
//station.adwAutoTip[1].04:=Cy_takeClamp2.xAutoTip;	   //Cy_takeClamp2 气缸自动中有手动
station.adwAutoTip[1].05:=Cy_takeClamp3.xAutoTip;	   //Cy_takeClamp3 气缸自动中有手动
//station.adwAutoTip[1].06:=Cy_takeClamp4.xAutoTip;	   //Cy_takeClamp4 气缸自动中有手动
station.adwAutoTip[1].07:=Cy_lifter	.xAutoTip;	     //Cy_lifter 气缸自动中有手动
END_ACTION

ACTION FlowInit:
IF NOT station.xIniting THEN
  station.iStepInit:=0;    
ELSE
//--------------------------------------------初始化步序----------------------------------
CASE station.iStepInit OF	
 0://  
  	IF station.xIniting THEN	
  	  station.iStepInit:=10;	
  	END_IF	
10://复位数据
    CardState[1].Card_OK:=FALSE;
 	  CardState[1].A:=FALSE;
	  CardState[1].B:=FALSE;
    station.iStepInit := 20 ;		
20://升降气缸原点
    Cy_lifter.xInit := TRUE ;
		IF Cy_lifter.xHP_Delay   
    THEN 
    station.iStepInit:=30;	
		END_IF
30://气缸回原点
    Cy_rotate.xInit := TRUE ;
		IF Cy_rotate.xHP_Delay THEN
			Cy_takeClamp1.xInit:=TRUE;
	//		Cy_takeClamp2.xInit:=TRUE;
			Cy_takeClamp3.xInit:=TRUE;
	//		Cy_takeClamp4.xInit:=TRUE;
		END_IF
    IF Cy_takeClamp1.xHP_Delay //AND Cy_takeClamp2.xHP_Delay 
			AND Cy_takeClamp3.xHP_Delay //AND Cy_takeClamp4.xHP_Delay
			AND Cy_rotate.xHP_Delay AND  Cy_lifter.xHP_Delay
THEN 
    station.iStepInit:=999;	
		END_IF
		
999://初始化完成	
	station.iStepInit:=0;
	station.xInitDone:=TRUE;  
END_CASE
END_IF
END_ACTION

ACTION ILC:

//---------------------------------------------------工站可执行-------------------------------------------------------
station.xCanRun := TRUE ;

//---------------------------------------------------气缸动作条件-------------------------------------------
Cy_rotate.xOnILC:=Cy_lifter.xHP_Sensor OR Cy_rotate.xWP_Valve;
Cy_rotate.xOffILC:=Cy_lifter.xHP_Sensor OR Cy_rotate.xHP_Valve;

Cy_takeClamp1.xOnILC:=
Cy_takeClamp1.xOffILC:=TRUE;
                       //Cy_lifter.xWP_Delay 

//Cy_takeClamp2.xOnILC:=
//Cy_takeClamp2.xOffILC:=TRUE;

Cy_takeClamp3.xOnILC:=
Cy_takeClamp3.xOffILC:=TRUE;


//Cy_takeClamp4.xOnILC:=
//Cy_takeClamp4.xOffILC:=TRUE;

Cy_lifter.xOnILC:=NOT S05_CircleLine.Axis_Cycleline.xbusy AND Cy_rotate_on;
Cy_lifter.xOffILC:= TRUE ;
END_ACTION

ACTION FlowAuto:

//-----------------------------------------初始化是否完成判断----------------------------------------------
IF NOT station.xInitDone 
THEN
 	station.iStepAuto:=0;
 	station.xDone:=FALSE;
ELSIF station.xRunning 
THEN
//-----------------------------------------动作步骤--------------------------------------------------------
CASE station.iStepAuto OF	  
	0: //----Home Step，等待启动----
		
